C03663=1120.671,285.991,-75.029,-178.079,10.307,149.546
C03664=1120.667,286.239,-75.060,-178.076,10.310,149.546
C03665=1120.663,286.487,-75.091,-178.074,10.312,149.545
C03666=1120.659,286.735,-75.121,-178.070,10.314,149.545
C03667=1120.655,286.984,-75.152,-178.067,10.317,149.545
C03668=1120.650,287.231,-75.183,-178.064,10.319,149.545
C03669=1120.646,287.479,-75.215,-178.061,10.322,149.545
C03670=1120.643,287.727,-75.245,-178.058,10.325,149.545
C03671=1120.638,287.975,-75.276,-178.055,10.327,149.544
C03672=1120.634,288.224,-75.307,-178.052,10.330,149.544
C03673=1120.629,288.472,-75.338,-178.048,10.332,149.544
C03674=1120.625,288.719,-75.368,-178.045,10.335,149.544
C03675=1120.622,288.967,-75.400,-178.043,10.337,149.544
C03676=1120.617,289.215,-75.431,-178.040,10.340,149.544
C03677=1120.613,289.464,-75.462,-178.036,10.342,149.543
C03678=1120.608,289.712,-75.493,-178.034,10.345,149.543
C03679=1120.605,289.959,-75.523,-178.030,10.347,149.543
C03680=1120.601,290.208,-75.555,-178.027,10.350,149.543
C03681=1120.596,290.456,-75.585,-178.024,10.353,149.543
C03682=1120.593,290.704,-75.617,-178.021,10.355,149.542
C03683=1120.588,290.952,-75.648,-178.018,10.358,149.542
C03684=1120.584,291.200,-75.679,-178.015,10.360,149.542
C03685=1120.580,291.447,-75.710,-178.012,10.362,149.542
C03686=1120.576,291.696,-75.741,-178.009,10.365,149.542
C03687=1120.572,291.944,-75.772,-178.006,10.368,149.542
C03688=1120.568,292.192,-75.804,-178.003,10.370,149.541
C03689=1120.563,292.440,-75.834,-178.000,10.373,149.541
C03690=1120.559,292.689,-75.866,-177.997,10.375,149.541
C03691=1120.555,292.936,-75.897,-177.994,10.378,149.541
C03692=1120.551,293.185,-75.928,-177.991,10.381,149.541
C03693=1120.547,293.432,-75.960,-177.987,10.383,149.541
C03694=1120.544,293.645,-75.986,-177.985,10.385,149.540
C03695=1120.540,293.858,-76.013,-177.983,10.387,149.540
C03696=1120.536,294.071,-76.040,-177.979,10.390,149.540
C03697=1120.533,294.283,-76.067,-177.977,10.392,149.540
C03698=1120.529,294.497,-76.094,-177.975,10.394,149.540
C03699=1120.526,294.710,-76.121,-177.971,10.396,149.540
C03700=1120.522,294.923,-76.147,-177.969,10.398,149.539
C03701=1120.519,295.135,-76.174,-177.967,10.400,149.539
C03702=1120.515,295.383,-76.206,-177.964,10.402,149.539
C03703=1120.511,295.632,-76.237,-177.961,10.405,149.539
C03704=1120.507,295.879,-76.268,-177.957,10.408,149.539
C03705=1120.503,296.128,-76.300,-177.954,10.410,149.539
C03706=1120.498,296.375,-76.331,-177.951,10.413,149.539
C03707=1120.495,296.623,-76.363,-177.948,10.415,149.538
C03708=1120.490,296.871,-76.394,-177.945,10.418,149.538
C03709=1120.486,297.119,-76.426,-177.942,10.421,149.538
C03710=1120.482,297.367,-76.458,-177.939,10.423,149.538
C03711=1120.477,297.615,-76.489,-177.936,10.425,149.538
C03712=1120.474,297.863,-76.521,-177.933,10.428,149.537
C03713=1120.469,298.111,-76.552,-177.930,10.430,149.537
C03714=1120.466,298.359,-76.584,-177.927,10.433,149.537
C03715=1120.462,298.608,-76.615,-177.924,10.435,149.537
C03716=1120.457,298.855,-76.646,-177.921,10.438,149.537
C03717=1120.454,299.103,-76.678,-177.917,10.441,149.536
C03718=1120.448,299.351,-76.710,-177.914,10.443,149.536
C03719=1120.444,299.599,-76.742,-177.911,10.446,149.536
C03720=1120.441,299.847,-76.773,-177.908,10.449,149.536
C03721=1120.436,300.095,-76.805,-177.905,10.451,149.536
C03722=1120.433,300.343,-76.837,-177.903,10.453,149.536
C03723=1120.429,300.591,-76.869,-177.899,10.456,149.535
C03724=1120.424,300.838,-76.901,-177.896,10.458,149.535
C03725=1120.420,301.086,-76.932,-177.893,10.461,149.535
C03726=1120.416,301.335,-76.964,-177.890,10.463,149.535
C03727=1120.412,301.582,-76.995,-177.887,10.466,149.535
C03728=1120.408,301.831,-77.028,-177.884,10.469,149.535
C03729=1120.404,302.079,-77.059,-177.880,10.471,149.534
C03730=1120.400,302.326,-77.091,-177.877,10.474,149.534
C03731=1120.396,302.574,-77.123,-177.874,10.476,149.534
C03732=1120.391,302.822,-77.155,-177.871,10.479,149.534
C03733=1120.387,303.070,-77.187,-177.868,10.481,149.534
C03734=1120.383,303.318,-77.218,-177.865,10.483,149.533
C03735=1120.379,303.566,-77.251,-177.862,10.486,149.533
C03736=1120.375,303.814,-77.283,-177.859,10.488,149.533
C03737=1120.371,304.062,-77.314,-177.856,10.491,149.533
C03738=1120.366,304.310,-77.347,-177.853,10.494,149.533
C03739=1120.363,304.558,-77.379,-177.850,10.496,149.533
C03740=1120.359,304.805,-77.411,-177.846,10.499,149.532
C03741=1120.354,305.053,-77.443,-177.843,10.502,149.532
C03742=1120.351,305.301,-77.475,-177.840,10.504,149.532
C03743=1120.346,305.549,-77.507,-177.837,10.507,149.532
C03744=1120.342,305.797,-77.539,-177.834,10.509,149.532
C03745=1120.338,306.045,-77.571,-177.832,10.511,149.532
C03746=1120.334,306.293,-77.603,-177.828,10.514,149.531
C03747=1120.330,306.541,-77.636,-177.825,10.516,149.531
C03748=1120.326,306.789,-77.668,-177.822,10.519,149.531
C03749=1120.322,307.036,-77.700,-177.819,10.521,149.531
C03750=1120.318,307.249,-77.727,-177.816,10.523,149.531
C03751=1120.315,307.462,-77.754,-177.813,10.526,149.531
C03752=1120.311,307.675,-77.783,-177.811,10.528,149.530
C03753=1120.308,307.887,-77.811,-177.808,10.530,149.530
C03754=1120.304,308.100,-77.838,-177.805,10.532,149.530
C03755=1120.301,308.313,-77.865,-177.803,10.534,149.530
C03756=1120.297,308.526,-77.893,-177.800,10.537,149.530
C03757=1120.294,308.738,-77.921,-177.798,10.539,149.530
C03758=1120.290,308.986,-77.953,-177.794,10.541,149.529
C03759=1120.285,309.235,-77.986,-177.791,10.544,149.529
C03760=1120.282,309.482,-78.018,-177.788,10.546,149.529
C03761=1120.278,309.730,-78.051,-177.785,10.549,149.529
C03762=1120.274,309.978,-78.083,-177.782,10.552,149.529
C03763=1120.270,310.226,-78.116,-177.779,10.553,149.528
C03764=1120.265,310.474,-78.148,-177.776,10.556,149.528
C03765=1120.261,310.721,-78.180,-177.773,10.559,149.528
C03766=1120.257,310.970,-78.213,-177.770,10.561,149.528
C03767=1120.253,311.217,-78.245,-177.766,10.564,149.528
C03768=1120.249,311.465,-78.278,-177.764,10.567,149.528
C03769=1120.246,311.713,-78.310,-177.760,10.569,149.527
C03770=1120.241,311.961,-78.343,-177.757,10.571,149.527
C03771=1120.237,312.209,-78.376,-177.754,10.574,149.527
C03772=1120.233,312.457,-78.408,-177.751,10.577,149.527
C03773=1120.229,312.704,-78.441,-177.748,10.579,149.527
C03774=1120.224,312.952,-78.473,-177.744,10.582,149.526
C03775=1120.221,313.200,-78.506,-177.742,10.583,149.526
C03776=1120.217,313.447,-78.539,-177.739,10.586,149.526
C03777=1120.213,313.696,-78.571,-177.735,10.589,149.526
C03778=1120.209,313.943,-78.604,-177.733,10.591,149.526
C03779=1120.204,314.192,-78.636,-177.729,10.594,149.526
C03780=1120.201,314.439,-78.669,-177.726,10.597,149.525
C03781=1120.197,314.687,-78.702,-177.723,10.599,149.525
C03782=1120.192,314.935,-78.734,-177.720,10.602,149.525
C03783=1120.188,315.183,-78.767,-177.717,10.604,149.525
C03784=1120.185,315.430,-78.800,-177.713,10.607,149.525
C03785=1120.181,315.678,-78.833,-177.710,10.610,149.525
C03786=1120.176,315.926,-78.866,-177.707,10.612,149.524
C03787=1120.173,316.174,-78.898,-177.704,10.614,149.524
C03788=1120.169,316.421,-78.931,-177.701,10.616,149.524
C03789=1120.165,316.669,-78.965,-177.698,10.619,149.524
C03790=1120.160,316.918,-78.997,-177.695,10.621,149.523
C03791=1120.157,317.165,-79.030,-177.692,10.624,149.523
C03792=1120.153,317.413,-79.063,-177.689,10.627,149.523
C03793=1120.148,317.660,-79.096,-177.686,10.629,149.523
C03794=1120.144,317.908,-79.129,-177.682,10.632,149.523
C03795=1120.140,318.156,-79.162,-177.679,10.634,149.523
C03796=1120.136,318.404,-79.194,-177.676,10.637,149.522
C03797=1120.132,318.652,-79.227,-177.673,10.639,149.522
C03798=1120.128,318.899,-79.260,-177.670,10.642,149.522
C03799=1120.124,319.147,-79.293,-177.666,10.645,149.522
C03800=1120.120,319.395,-79.327,-177.664,10.646,149.522
C03801=1120.116,319.643,-79.360,-177.661,10.649,149.522
C03802=1120.112,319.891,-79.393,-177.658,10.652,149.521
C03803=1120.109,320.138,-79.426,-177.654,10.654,149.521
C03804=1120.105,320.386,-79.459,-177.651,10.657,149.521
C03805=1120.101,320.634,-79.492,-177.648,10.659,149.521
C03806=1120.097,320.847,-79.521,-177.646,10.661,149.521
C03807=1120.094,321.059,-79.549,-177.642,10.664,149.520
C03808=1120.090,321.272,-79.578,-177.640,10.666,149.520
C03809=1120.087,321.484,-79.607,-177.637,10.668,149.520
C03810=1120.083,321.698,-79.634,-177.634,10.670,149.520
C03811=1120.079,321.910,-79.663,-177.632,10.672,149.520
C03812=1120.077,322.122,-79.691,-177.629,10.674,149.520
C03813=1120.073,322.335,-79.720,-177.627,10.676,149.520
C03814=1120.069,322.583,-79.753,-177.623,10.679,149.519
C03815=1120.065,322.831,-79.786,-177.620,10.682,149.519
C03816=1120.061,323.078,-79.820,-177.617,10.684,149.519
C03817=1120.057,323.325,-79.853,-177.614,10.687,149.519
C03818=1120.053,323.574,-79.887,-177.611,10.689,149.519
C03819=1120.049,323.822,-79.920,-177.607,10.692,149.518
C03820=1120.045,324.069,-79.953,-177.604,10.694,149.518
C03821=1120.041,324.316,-79.987,-177.602,10.696,149.518
C03822=1120.037,324.564,-80.020,-177.598,10.699,149.518
C03823=1120.033,324.813,-80.054,-177.595,10.701,149.518
C03824=1120.029,325.060,-80.087,-177.592,10.704,149.518
C03825=1120.026,325.307,-80.121,-177.589,10.706,149.517
C03826=1120.021,325.555,-80.154,-177.586,10.709,149.517
C03827=1120.017,325.803,-80.187,-177.583,10.712,149.517
C03828=1120.014,326.051,-80.221,-177.579,10.714,149.517
C03829=1120.009,326.299,-80.255,-177.576,10.716,149.516
C03830=1120.005,326.547,-80.288,-177.573,10.719,149.516
C03831=1120.001,326.794,-80.321,-177.570,10.722,149.516
C03832=1119.997,327.041,-80.355,-177.566,10.724,149.516
C03833=1119.993,327.290,-80.389,-177.563,10.727,149.516
C03834=1119.990,327.537,-80.423,-177.561,10.729,149.516
C03835=1119.986,327.785,-80.456,-177.557,10.731,149.515
C03836=1119.981,328.033,-80.490,-177.555,10.734,149.515
C03837=1119.977,328.280,-80.524,-177.551,10.736,149.515
C03838=1119.973,328.528,-80.557,-177.548,10.739,149.515
C03839=1119.969,328.775,-80.591,-177.545,10.741,149.515
C03840=1119.965,329.023,-80.624,-177.542,10.744,149.514
C03841=1119.961,329.271,-80.659,-177.538,10.746,149.514
C03842=1119.957,329.519,-80.692,-177.535,10.749,149.514
C03843=1119.953,329.766,-80.726,-177.532,10.752,149.514
C03844=1119.950,330.014,-80.759,-177.529,10.754,149.514
C03845=1119.945,330.262,-80.794,-177.525,10.757,149.513
C03846=1119.941,330.509,-80.828,-177.523,10.759,149.513
C03847=1119.937,330.757,-80.861,-177.519,10.762,149.513
C03848=1119.934,331.005,-80.895,-177.517,10.763,149.513
C03849=1119.929,331.253,-80.929,-177.513,10.766,149.513
C03850=1119.925,331.500,-80.963,-177.510,10.769,149.513
C03851=1119.922,331.747,-80.997,-177.507,10.771,149.512
C03852=1119.918,331.995,-81.030,-177.504,10.774,149.512
C03853=1119.913,332.243,-81.065,-177.501,10.776,149.512
C03854=1119.910,332.490,-81.099,-177.497,10.779,149.512
C03855=1119.906,332.738,-81.132,-177.494,10.781,149.512
C03856=1119.902,332.986,-81.167,-177.491,10.784,149.511
C03857=1119.898,333.233,-81.201,-177.488,10.786,149.511
C03858=1119.893,333.481,-81.234,-177.485,10.789,149.511
C03859=1119.890,333.729,-81.269,-177.481,10.791,149.511
C03860=1119.886,333.976,-81.303,-177.478,10.794,149.511
C03861=1119.882,334.224,-81.337,-177.475,10.797,149.510
C03862=1119.878,334.437,-81.366,-177.472,10.798,149.510
C03863=1119.875,334.649,-81.395,-177.470,10.800,149.510
C03864=1119.872,334.861,-81.425,-177.467,10.803,149.510
C03865=1119.868,335.074,-81.454,-177.464,10.805,149.510
C03866=1119.865,335.286,-81.484,-177.462,10.806,149.510
C03867=1119.862,335.499,-81.512,-177.459,10.809,149.509
C03868=1119.858,335.711,-81.542,-177.456,10.811,149.509
C03869=1119.855,335.924,-81.572,-177.454,10.813,149.509
C03870=1119.852,336.172,-81.605,-177.450,10.815,149.509
C03871=1119.847,336.420,-81.640,-177.447,10.818,149.509
C03872=1119.843,336.667,-81.673,-177.444,10.820,149.508
C03873=1119.839,336.915,-81.708,-177.441,10.823,149.508
C03874=1119.835,337.162,-81.742,-177.438,10.825,149.508
C03875=1119.831,337.410,-81.777,-177.434,10.828,149.508
C03876=1119.828,337.657,-81.811,-177.431,10.830,149.508
C03877=1119.824,337.905,-81.846,-177.428,10.833,149.508
C03878=1119.820,338.152,-81.880,-177.425,10.836,149.507
C03879=1119.816,338.400,-81.914,-177.421,10.838,149.507
C03880=1119.812,338.648,-81.948,-177.418,10.841,149.507
C03881=1119.808,338.896,-81.983,-177.415,10.843,149.507
C03882=1119.804,339.143,-82.017,-177.412,10.846,149.507
C03883=1119.800,339.391,-82.052,-177.409,10.847,149.506
C03884=1119.796,339.638,-82.086,-177.406,10.850,149.506
C03885=1119.793,339.886,-82.121,-177.403,10.852,149.506
C03886=1119.788,340.133,-82.156,-177.400,10.855,149.506
C03887=1119.784,340.381,-82.191,-177.396,10.858,149.506
C03888=1119.780,340.628,-82.224,-177.393,10.860,149.505
C03889=1119.776,340.876,-82.259,-177.390,10.863,149.505
C03890=1119.773,341.123,-82.293,-177.386,10.865,149.505
C03891=1119.769,341.371,-82.329,-177.383,10.868,149.505
C03892=1119.764,341.618,-82.363,-177.380,10.870,149.505
C03893=1119.761,341.866,-82.397,-177.377,10.873,149.504
C03894=1119.756,342.114,-82.432,-177.374,10.875,149.504
C03895=1119.753,342.362,-82.467,-177.370,10.878,149.504
C03896=1119.748,342.608,-82.502,-177.367,10.880,149.504
C03897=1119.745,342.856,-82.536,-177.364,10.883,149.504
C03898=1119.740,343.104,-82.571,-177.361,10.885,149.503
C03899=1119.737,343.351,-82.606,-177.358,10.887,149.503
C03900=1119.734,343.599,-82.640,-177.355,10.889,149.503
C03901=1119.729,343.846,-82.675,-177.352,10.892,149.503
C03902=1119.725,344.094,-82.710,-177.348,10.895,149.503
C03903=1119.721,344.341,-82.745,-177.345,10.897,149.502
C03904=1119.718,344.589,-82.779,-177.342,10.900,149.502
C03905=1119.714,344.837,-82.815,-177.338,10.902,149.502
C03906=1119.709,345.084,-82.849,-177.335,10.904,149.502
C03907=1119.706,345.332,-82.885,-177.332,10.907,149.502
C03908=1119.701,345.579,-82.919,-177.329,10.910,149.501
C03909=1119.698,345.826,-82.954,-177.326,10.912,149.501
C03910=1119.694,346.074,-82.989,-177.322,10.915,149.501
C03911=1119.690,346.322,-83.023,-177.319,10.917,149.501
C03912=1119.686,346.569,-83.059,-177.316,10.919,149.500
C03913=1119.682,346.817,-83.094,-177.313,10.922,149.500
C03914=1119.678,347.064,-83.129,-177.310,10.924,149.500
C03915=1119.675,347.311,-83.164,-177.307,10.927,149.500
C03916=1119.671,347.559,-83.199,-177.303,10.929,149.500
C03917=1119.667,347.806,-83.234,-177.300,10.931,149.500
C03918=1119.663,348.020,-83.264,-177.298,10.933,149.499
C03919=1119.660,348.232,-83.294,-177.295,10.936,149.499
C03920=1119.657,348.444,-83.324,-177.292,10.938,149.499
C03921=1119.653,348.656,-83.355,-177.289,10.940,149.499
C03922=1119.650,348.868,-83.384,-177.286,10.942,149.499
C03923=1119.646,349.081,-83.414,-177.284,10.944,149.499
C03924=1119.644,349.293,-83.445,-177.281,10.947,149.498
C03925=1119.640,349.506,-83.475,-177.278,10.948,149.498
C03926=1119.636,349.753,-83.511,-177.275,10.951,149.498
C03927=1119.631,350.001,-83.545,-177.271,10.954,149.498
C03928=1119.628,350.248,-83.581,-177.267,10.956,149.497
C03929=1119.624,350.496,-83.616,-177.264,10.959,149.497
C03930=1119.621,350.743,-83.651,-177.261,10.961,149.497
C03931=1119.617,350.990,-83.686,-177.258,10.964,149.497
C03932=1119.613,351.238,-83.721,-177.254,10.966,149.497
C03933=1119.609,351.485,-83.757,-177.250,10.969,149.496
C03934=1119.606,351.733,-83.792,-177.247,10.972,149.496
C03935=1119.601,351.980,-83.828,-177.243,10.974,149.496
C03936=1119.597,352.228,-83.863,-177.240,10.977,149.495
C03937=1119.593,352.475,-83.899,-177.237,10.979,149.495
C03938=1119.589,352.723,-83.934,-177.233,10.981,149.495
C03939=1119.586,352.970,-83.970,-177.229,10.985,149.495
C03940=1119.581,353.217,-84.005,-177.226,10.987,149.495
C03941=1119.578,353.465,-84.040,-177.222,10.989,149.494
C03942=1119.574,353.712,-84.076,-177.219,10.992,149.494
C03943=1119.570,353.960,-84.111,-177.216,10.994,149.494
C03944=1119.567,354.207,-84.147,-177.212,10.997,149.494
C03945=1119.563,354.454,-84.182,-177.209,10.999,149.493
C03946=1119.559,354.702,-84.218,-177.206,11.002,149.493
C03947=1119.555,354.949,-84.253,-177.202,11.004,149.493
C03948=1119.551,355.197,-84.289,-177.198,11.007,149.493
C03949=1119.547,355.444,-84.325,-177.195,11.009,149.492
C03950=1119.543,355.692,-84.361,-177.192,11.012,149.492
C03951=1119.540,355.939,-84.396,-177.188,11.014,149.492
C03952=1119.536,356.186,-84.431,-177.185,11.017,149.491
C03953=1119.532,356.434,-84.467,-177.181,11.019,149.491
C03954=1119.527,356.681,-84.503,-177.178,11.021,149.491
C03955=1119.524,356.929,-84.538,-177.175,11.024,149.491
C03956=1119.520,357.176,-84.574,-177.171,11.026,149.491
C03957=1119.517,357.423,-84.610,-177.168,11.029,149.490
C03958=1119.513,357.671,-84.646,-177.164,11.031,149.490
C03959=1119.509,357.919,-84.682,-177.161,11.033,149.490
C03960=1119.505,358.166,-84.718,-177.158,11.036,149.490
C03961=1119.501,358.414,-84.753,-177.154,11.038,149.489
C03962=1119.498,358.661,-84.789,-177.151,11.041,149.489
C03963=1119.494,358.908,-84.825,-177.147,11.043,149.489
C03964=1119.489,359.155,-84.861,-177.144,11.045,149.488
C03965=1119.486,359.403,-84.896,-177.141,11.048,149.488
C03966=1119.482,359.650,-84.932,-177.137,11.050,149.488
C03967=1119.478,359.897,-84.969,-177.134,11.053,149.488
C03968=1119.474,360.145,-85.004,-177.130,11.055,149.487
C03969=1119.471,360.392,-85.040,-177.127,11.057,149.487
C03970=1119.467,360.640,-85.077,-177.123,11.060,149.487
C03971=1119.463,360.887,-85.112,-177.120,11.062,149.487
C03972=1119.460,361.134,-85.148,-177.117,11.065,149.486
C03973=1119.455,361.382,-85.185,-177.114,11.067,149.486
C03974=1119.452,361.594,-85.216,-177.110,11.069,149.486
C03975=1119.449,361.806,-85.246,-177.108,11.071,149.486
C03976=1119.446,362.019,-85.277,-177.104,11.074,149.485
C03977=1119.442,362.231,-85.308,-177.102,11.075,149.485
C03978=1119.439,362.443,-85.339,-177.098,11.078,149.485
C03979=1119.436,362.655,-85.370,-177.096,11.079,149.485
C03980=1119.433,362.867,-85.401,-177.093,11.081,149.485
C03981=1119.430,363.079,-85.432,-177.090,11.084,149.484
C03982=1119.426,363.327,-85.469,-177.086,11.086,149.484
C03983=1119.422,363.574,-85.505,-177.083,11.089,149.484
C03984=1119.418,363.821,-85.541,-177.080,11.091,149.484
C03985=1119.415,364.068,-85.578,-177.076,11.094,149.483
C03986=1119.411,364.316,-85.613,-177.073,11.096,149.483
C03987=1119.407,364.563,-85.650,-177.070,11.097,149.483
C03988=1119.403,364.810,-85.686,-177.067,11.100,149.483
C03989=1119.399,365.058,-85.722,-177.063,11.102,149.482
C03990=1119.396,365.304,-85.759,-177.060,11.105,149.482
C03991=1119.392,365.553,-85.795,-177.057,11.107,149.482
C03992=1119.389,365.800,-85.831,-177.054,11.110,149.482
C03993=1119.385,366.047,-85.868,-177.050,11.112,149.481
C03994=1119.380,366.295,-85.904,-177.047,11.114,149.481
C03995=1119.377,366.542,-85.941,-177.043,11.117,149.481
C03996=1119.373,366.789,-85.978,-177.040,11.119,149.481
C03997=1119.369,367.036,-86.014,-177.037,11.122,149.480
C03998=1119.365,367.284,-86.050,-177.033,11.124,149.480
C03999=1119.362,367.531,-86.086,-177.030,11.126,149.480
C04000=1119.357,367.778,-86.123,-177.026,11.129,149.480
C04001=1119.354,368.026,-86.160,-177.024,11.131,149.479
C04002=1119.350,368.273,-86.196,-177.020,11.133,149.479
C04003=1119.346,368.520,-86.233,-177.017,11.136,149.479
C04004=1119.342,368.768,-86.270,-177.014,11.138,149.479
C04005=1119.339,369.014,-86.306,-177.010,11.140,149.479
C04006=1119.335,369.262,-86.343,-177.007,11.143,149.478
C04007=1119.332,369.509,-86.379,-177.004,11.145,149.478
C04008=1119.328,369.756,-86.416,-177.001,11.148,149.478
C04009=1119.324,370.004,-86.453,-176.997,11.150,149.478
C04010=1119.320,370.250,-86.489,-176.994,11.153,149.477
C04011=1119.316,370.498,-86.525,-176.990,11.155,149.477
C04012=1119.312,370.745,-86.562,-176.988,11.157,149.477
C04013=1119.308,370.993,-86.600,-176.984,11.159,149.477
C04014=1119.305,371.240,-86.636,-176.981,11.162,149.476
C04015=1119.301,371.487,-86.673,-176.978,11.164,149.476
C04016=1119.297,371.735,-86.710,-176.974,11.167,149.476
C04017=1119.294,371.982,-86.746,-176.971,11.169,149.476
C04018=1119.290,372.229,-86.783,-176.968,11.172,149.476
C04019=1119.286,372.476,-86.821,-176.964,11.174,149.475
C04020=1119.282,372.723,-86.857,-176.961,11.177,149.475
C04021=1119.279,372.971,-86.894,-176.959,11.178,149.475
C04022=1119.275,373.218,-86.931,-176.955,11.181,149.475
C04023=1119.271,373.465,-86.968,-176.952,11.183,149.475
C04024=1119.267,373.712,-87.005,-176.949,11.186,149.475
C04025=1119.264,373.960,-87.042,-176.946,11.188,149.474
C04026=1119.260,374.207,-87.078,-176.942,11.191,149.474
C04027=1119.256,374.454,-87.116,-176.939,11.193,149.474
C04028=1119.252,374.701,-87.153,-176.936,11.196,149.474
C04029=1119.249,374.949,-87.190,-176.933,11.198,149.473
C04030=1119.245,375.160,-87.221,-176.930,11.200,149.473
C04031=1119.242,375.373,-87.253,-176.928,11.202,149.473
C04032=1119.239,375.585,-87.285,-176.925,11.204,149.473
C04033=1119.236,375.796,-87.317,-176.922,11.207,149.473
C04034=1119.233,376.009,-87.348,-176.919,11.208,149.473
C04035=1119.230,376.221,-87.380,-176.917,11.210,149.473
C04036=1119.226,376.433,-87.412,-176.914,11.213,149.472
C04037=1119.223,376.645,-87.444,-176.911,11.215,149.472
C04038=1119.219,376.892,-87.481,-176.908,11.217,149.472
C04039=1119.215,377.140,-87.518,-176.905,11.220,149.472
C04040=1119.212,377.386,-87.556,-176.902,11.222,149.472
C04041=1119.208,377.633,-87.593,-176.898,11.225,149.472
C04042=1119.204,377.881,-87.630,-176.896,11.227,149.472
C04043=1119.200,378.128,-87.668,-176.893,11.229,149.471
C04044=1119.196,378.375,-87.705,-176.889,11.232,149.471
C04045=1119.194,378.622,-87.742,-176.886,11.234,149.471
C04046=1119.190,378.869,-87.779,-176.883,11.237,149.471
C04047=1119.186,379.116,-87.816,-176.880,11.240,149.471
C04048=1119.182,379.364,-87.854,-176.877,11.242,149.471
C04049=1119.178,379.611,-87.890,-176.874,11.245,149.471
C04050=1119.175,379.858,-87.928,-176.871,11.247,149.470
C04051=1119.170,380.106,-87.966,-176.868,11.249,149.470
C04052=1119.166,380.352,-88.003,-176.865,11.252,149.470
C04053=1119.163,380.600,-88.041,-176.862,11.254,149.470
C04054=1119.159,380.847,-88.078,-176.859,11.257,149.470
C04055=1119.156,381.094,-88.116,-176.855,11.260,149.470
C04056=1119.152,381.341,-88.153,-176.853,11.262,149.470
C04057=1119.148,381.588,-88.191,-176.849,11.265,149.469
C04058=1119.145,381.836,-88.228,-176.847,11.267,149.469
C04059=1119.141,382.082,-88.265,-176.844,11.269,149.469
C04060=1119.138,382.330,-88.303,-176.841,11.272,149.469
C04061=1119.134,382.577,-88.340,-176.837,11.275,149.469
C04062=1119.130,382.824,-88.378,-176.835,11.278,149.469
C04063=1119.127,383.071,-88.416,-176.832,11.280,149.469
C04064=1119.122,383.319,-88.453,-176.828,11.283,149.469
C04065=1119.119,383.565,-88.491,-176.826,11.285,149.469
C04066=1119.115,383.812,-88.529,-176.824,11.287,149.469
C04067=1119.111,384.060,-88.566,-176.822,11.289,149.469
C04068=1119.107,384.306,-88.603,-176.820,11.291,149.469
C04069=1119.104,384.554,-88.641,-176.818,11.294,149.469
C04070=1119.101,384.800,-88.679,-176.816,11.296,149.469
C04071=1119.096,385.048,-88.717,-176.813,11.299,149.469
C04072=1119.092,385.295,-88.754,-176.811,11.301,149.469
C04073=1119.089,385.542,-88.792,-176.809,11.303,149.469
C04074=1119.086,385.789,-88.830,-176.807,11.305,149.469
C04075=1119.082,386.036,-88.868,-176.805,11.308,149.469
C04076=1119.077,386.284,-88.905,-176.803,11.310,149.469
C04077=1119.074,386.531,-88.943,-176.801,11.312,149.469
C04078=1119.071,386.777,-88.981,-176.799,11.314,149.469
C04079=1119.067,387.025,-89.019,-176.797,11.317,149.470
C04080=1119.064,387.272,-89.057,-176.794,11.320,149.470
C04081=1119.060,387.519,-89.095,-176.792,11.322,149.470
C04082=1119.056,387.767,-89.132,-176.790,11.324,149.470
C04083=1119.052,388.013,-89.170,-176.788,11.327,149.470
C04084=1119.049,388.261,-89.208,-176.786,11.329,149.470
C04085=1119.045,388.507,-89.246,-176.784,11.332,149.470
C04086=1119.042,388.719,-89.278,-176.783,11.334,149.470
C04087=1119.039,388.931,-89.311,-176.781,11.336,149.470
C04088=1119.036,389.143,-89.343,-176.779,11.338,149.471
C04089=1119.032,389.356,-89.376,-176.777,11.341,149.471
C04090=1119.030,389.567,-89.408,-176.776,11.343,149.471
C04091=1119.026,389.779,-89.441,-176.774,11.345,149.471
C04092=1119.023,389.990,-89.474,-176.773,11.347,149.471
C04093=1119.020,390.202,-89.506,-176.771,11.350,149.471
C04094=1119.017,390.450,-89.544,-176.769,11.352,149.472
C04095=1119.012,390.696,-89.582,-176.767,11.356,149.472
C04096=1119.009,390.944,-89.620,-176.765,11.358,149.472
C04097=1119.005,391.190,-89.657,-176.763,11.361,149.472
C04098=1119.001,391.438,-89.696,-176.761,11.364,149.473
C04099=1118.998,391.685,-89.734,-176.759,11.367,149.473
C04100=1118.994,391.932,-89.771,-176.758,11.369,149.473
C04101=1118.991,392.179,-89.810,-176.755,11.372,149.473
C04102=1118.987,392.427,-89.848,-176.754,11.375,149.474
C04103=1118.984,392.673,-89.886,-176.752,11.378,149.474
C04104=1118.980,392.920,-89.925,-176.750,11.381,149.474
C04105=1118.976,393.167,-89.962,-176.748,11.384,149.475
C04106=1118.972,393.414,-90.001,-176.746,11.387,149.475
C04107=1118.969,393.662,-90.039,-176.745,11.390,149.475
C04108=1118.965,393.908,-90.076,-176.743,11.393,149.476
C04109=1118.961,394.156,-90.115,-176.741,11.396,149.476
C04110=1118.958,394.403,-90.153,-176.740,11.399,149.476
C04111=1118.954,394.649,-90.192,-176.738,11.402,149.477
C04112=1118.951,394.896,-90.230,-176.737,11.405,149.477
C04113=1118.946,395.143,-90.268,-176.734,11.409,149.478
C04114=1118.943,395.391,-90.306,-176.732,11.412,149.478
C04115=1118.940,395.637,-90.344,-176.731,11.415,149.478
C04116=1118.936,395.884,-90.383,-176.729,11.418,149.479
C04117=1118.932,396.131,-90.421,-176.728,11.421,149.479
C04118=1118.929,396.379,-90.459,-176.726,11.425,149.480
C04119=1118.925,396.625,-90.497,-176.724,11.428,149.480
C04120=1118.921,396.873,-90.536,-176.723,11.431,149.481
C04121=1118.918,397.120,-90.574,-176.721,11.435,149.481
C04122=1118.914,397.367,-90.612,-176.720,11.438,149.481
C04123=1118.911,397.613,-90.651,-176.718,11.442,149.482
C04124=1118.907,397.861,-90.689,-176.716,11.445,149.482
C04125=1118.903,398.108,-90.727,-176.715,11.448,149.483
C04126=1118.899,398.354,-90.766,-176.713,11.452,149.483
C04127=1118.896,398.602,-90.804,-176.711,11.456,149.484
C04128=1118.892,398.849,-90.843,-176.710,11.459,149.484
C04129=1118.889,399.096,-90.881,-176.708,11.463,149.485
C04130=1118.885,399.343,-90.919,-176.707,11.466,149.486
C04131=1118.881,399.590,-90.959,-176.706,11.469,149.486
C04132=1118.878,399.837,-90.997,-176.704,11.473,149.487
C04133=1118.874,400.083,-91.035,-176.703,11.477,149.487
C04134=1118.870,400.331,-91.073,-176.701,11.481,149.488
C04135=1118.867,400.578,-91.113,-176.699,11.485,149.488
C04136=1118.864,400.825,-91.151,-176.698,11.488,149.489
C04137=1118.859,401.072,-91.189,-176.697,11.492,149.490
C04138=1118.856,401.319,-91.228,-176.695,11.496,149.490
C04139=1118.852,401.566,-91.266,-176.694,11.500,149.491
C04140=1118.849,401.813,-91.305,-176.692,11.504,149.492
C04141=1118.846,402.060,-91.344,-176.691,11.508,149.492
C04142=1118.842,402.272,-91.376,-176.690,11.511,149.493
C04143=1118.839,402.484,-91.410,-176.689,11.514,149.493
C04144=1118.836,402.695,-91.443,-176.687,11.518,149.494
C04145=1118.833,402.907,-91.476,-176.686,11.521,149.495
C04146=1118.830,403.119,-91.510,-176.685,11.525,149.495
C04147=1118.827,403.330,-91.542,-176.684,11.528,149.496
C04148=1118.824,403.542,-91.576,-176.683,11.532,149.497
C04149=1118.821,403.754,-91.609,-176.681,11.536,149.497
C04150=1118.816,404.000,-91.647,-176.681,11.540,149.498
C04151=1118.813,404.247,-91.686,-176.679,11.544,149.499
C04152=1118.810,404.494,-91.725,-176.678,11.548,149.500
C04153=1118.806,404.742,-91.764,-176.677,11.552,149.500
C04154=1118.802,404.989,-91.803,-176.676,11.557,149.501
C04155=1118.799,405.235,-91.841,-176.674,11.561,149.502
C04156=1118.795,405.482,-91.880,-176.673,11.565,149.503
C04157=1118.791,405.729,-91.919,-176.672,11.570,149.504
C04158=1118.788,405.976,-91.958,-176.671,11.574,149.505
C04159=1118.784,406.223,-91.996,-176.669,11.579,149.505
C04160=1118.781,406.470,-92.035,-176.668,11.583,149.506
C04161=1118.777,406.717,-92.075,-176.667,11.588,149.507
C04162=1118.774,406.963,-92.113,-176.666,11.592,149.508
C04163=1118.770,407.211,-92.151,-176.665,11.597,149.509
C04164=1118.766,407.458,-92.191,-176.664,11.602,149.510
C04165=1118.763,407.705,-92.230,-176.663,11.606,149.511
C04166=1118.760,407.951,-92.269,-176.662,11.611,149.512
C04167=1118.756,408.198,-92.308,-176.661,11.615,149.513
C04168=1118.752,408.446,-92.346,-176.659,11.620,149.514
C04169=1118.749,408.693,-92.386,-176.659,11.625,149.515
C04170=1118.746,408.940,-92.424,-176.658,11.630,149.516
C04171=1118.741,409.186,-92.463,-176.657,11.635,149.517
C04172=1118.738,409.433,-92.502,-176.656,11.640,149.518
C04173=1118.734,409.680,-92.542,-176.655,11.644,149.519
C04174=1118.731,409.927,-92.581,-176.654,11.650,149.520
C04175=1118.727,410.174,-92.620,-176.653,11.654,149.521
C04176=1118.724,410.420,-92.659,-176.652,11.659,149.522
C04177=1118.720,410.668,-92.697,-176.651,11.665,149.523
C04178=1118.717,410.915,-92.737,-176.650,11.669,149.524
C04179=1118.713,411.162,-92.776,-176.649,11.675,149.525
C04180=1118.709,411.409,-92.815,-176.648,11.680,149.527
C04181=1118.706,411.656,-92.854,-176.648,11.685,149.528
C04182=1118.702,411.903,-92.894,-176.647,11.690,149.529
C04183=1118.699,412.149,-92.932,-176.646,11.696,149.530
C04184=1118.696,412.396,-92.971,-176.645,11.701,149.531
C04185=1118.692,412.643,-93.011,-176.645,11.706,149.533
C04186=1118.688,412.890,-93.050,-176.643,11.712,149.534
C04187=1118.684,413.136,-93.089,-176.643,11.717,149.535
C04188=1118.681,413.383,-93.129,-176.642,11.723,149.536
C04189=1118.677,413.630,-93.168,-176.642,11.728,149.537
C04190=1118.675,413.877,-93.207,-176.641,11.734,149.539
C04191=1118.671,414.124,-93.246,-176.640,11.739,149.540
C04192=1118.670,414.371,-93.285,-176.640,11.744,149.541
C04193=1118.668,414.618,-93.324,-176.639,11.750,149.543
C04194=1118.667,414.864,-93.364,-176.638,11.756,149.544
C04195=1118.666,415.112,-93.402,-176.637,11.762,149.545
C04196=1118.666,415.359,-93.441,-176.637,11.767,149.547
C04197=1118.667,415.606,-93.480,-176.636,11.773,149.548
C04198=1118.668,415.818,-93.513,-176.636,11.778,149.549
C04199=1118.669,416.028,-93.546,-176.636,11.783,149.550
C04200=1118.671,416.240,-93.579,-176.635,11.788,149.552
C04201=1118.673,416.452,-93.612,-176.635,11.793,149.553
C04202=1118.675,416.663,-93.645,-176.635,11.798,149.554
C04203=1118.678,416.875,-93.678,-176.634,11.803,149.555
C04204=1118.682,417.086,-93.711,-176.634,11.808,149.556
C04205=1118.686,417.298,-93.744,-176.634,11.813,149.558
C04206=1118.267,417.298,-93.806,-176.626,11.818,149.557
C04207=1118.263,417.086,-93.774,-176.626,11.813,149.556
C04208=1118.259,416.874,-93.741,-176.627,11.807,149.555
C04209=1118.256,416.663,-93.708,-176.627,11.802,149.553
C04210=1118.254,416.452,-93.675,-176.628,11.797,149.552
C04211=1118.252,416.240,-93.642,-176.628,11.792,149.551
C04212=1118.250,416.028,-93.609,-176.628,11.787,149.550
C04213=1118.249,415.818,-93.576,-176.629,11.782,149.549
C04214=1118.248,415.605,-93.542,-176.629,11.777,149.547
C04215=1118.248,415.359,-93.503,-176.630,11.772,149.546
C04216=1118.247,415.112,-93.465,-176.631,11.766,149.545
C04217=1118.247,414.865,-93.426,-176.632,11.760,149.543
C04218=1118.249,414.618,-93.387,-176.632,11.755,149.542
C04219=1118.250,414.370,-93.347,-176.633,11.749,149.541
C04220=1118.252,414.124,-93.309,-176.633,11.743,149.539
C04221=1118.255,413.877,-93.269,-176.634,11.737,149.538
C04222=1118.258,413.630,-93.230,-176.635,11.732,149.537
C04223=1118.262,413.383,-93.191,-176.636,11.726,149.536
C04224=1118.265,413.136,-93.152,-176.636,11.721,149.534
C04225=1118.269,412.890,-93.112,-176.637,11.716,149.533
C04226=1118.272,412.643,-93.073,-176.638,11.710,149.532
C04227=1118.276,412.396,-93.034,-176.639,11.704,149.531
C04228=1118.280,412.149,-92.995,-176.640,11.700,149.530
C04229=1118.283,411.902,-92.955,-176.641,11.694,149.528
C04230=1118.287,411.655,-92.916,-176.641,11.689,149.527
C04231=1118.290,411.408,-92.877,-176.643,11.684,149.526
C04232=1118.293,411.161,-92.838,-176.644,11.678,149.525
C04233=1118.297,410.914,-92.799,-176.644,11.673,149.524
C04234=1118.301,410.667,-92.760,-176.645,11.668,149.523
C04235=1118.304,410.420,-92.720,-176.646,11.663,149.522
C04236=1118.308,410.173,-92.681,-176.647,11.658,149.520
C04237=1118.312,409.927,-92.642,-176.648,11.653,149.520
C04238=1118.315,409.680,-92.604,-176.649,11.648,149.518
C04239=1118.319,409.433,-92.564,-176.650,11.643,149.517
C04240=1118.322,409.186,-92.525,-176.651,11.638,149.516
C04241=1118.326,408.939,-92.486,-176.652,11.633,149.515
C04242=1118.329,408.692,-92.447,-176.653,11.628,149.514
C04243=1118.333,408.445,-92.409,-176.655,11.623,149.513
C04244=1118.336,408.198,-92.369,-176.656,11.619,149.512
C04245=1118.340,407.951,-92.330,-176.657,11.614,149.511
C04246=1118.343,407.704,-92.291,-176.658,11.609,149.510
C04247=1118.347,407.457,-92.252,-176.659,11.605,149.510
C04248=1118.351,407.211,-92.213,-176.660,11.600,149.509
C04249=1118.355,406.964,-92.175,-176.661,11.596,149.508
C04250=1118.358,406.717,-92.136,-176.663,11.590,149.507
C04251=1118.362,406.470,-92.096,-176.663,11.586,149.506
C04252=1118.365,406.223,-92.058,-176.665,11.582,149.505
C04253=1118.369,405.976,-92.019,-176.666,11.577,149.504
C04254=1118.372,405.729,-91.980,-176.667,11.573,149.503
C04255=1118.376,405.482,-91.941,-176.669,11.568,149.502
C04256=1118.379,405.236,-91.902,-176.670,11.564,149.502
C04257=1118.383,404.988,-91.864,-176.671,11.560,149.501
C04258=1118.387,404.741,-91.825,-176.672,11.555,149.500
C04259=1118.390,404.495,-91.786,-176.673,11.551,149.499
C04260=1118.394,404.247,-91.747,-176.675,11.547,149.498
C04261=1118.398,404.001,-91.709,-176.676,11.543,149.498
C04262=1118.401,403.754,-91.670,-176.677,11.539,149.497
C04263=1118.404,403.542,-91.637,-176.679,11.534,149.496
C04264=1118.407,403.331,-91.603,-176.680,11.531,149.496
C04265=1118.411,403.118,-91.571,-176.681,11.527,149.495
C04266=1118.414,402.907,-91.537,-176.682,11.524,149.494
C04267=1118.417,402.695,-91.504,-176.683,11.520,149.494
C04268=1118.419,402.484,-91.471,-176.684,11.517,149.493
C04269=1118.422,402.272,-91.438,-176.686,11.514,149.493
C04270=1118.426,402.060,-91.405,-176.687,11.510,149.492
C04271=1118.429,401.813,-91.366,-176.689,11.506,149.491
C04272=1118.432,401.566,-91.328,-176.690,11.502,149.491
C04273=1118.436,401.319,-91.288,-176.691,11.498,149.490
C04274=1118.441,401.072,-91.250,-176.693,11.494,149.489
C04275=1118.443,400.825,-91.211,-176.694,11.491,149.489
C04276=1118.447,400.578,-91.173,-176.695,11.487,149.488
C04277=1118.450,400.331,-91.134,-176.697,11.483,149.488
C04278=1118.455,400.084,-91.096,-176.699,11.479,149.487
C04279=1118.459,399.837,-91.058,-176.700,11.475,149.486
C04280=1118.462,399.590,-91.019,-176.702,11.472,149.486
C04281=1118.466,399.342,-90.980,-176.703,11.469,149.485
C04282=1118.469,399.097,-90.942,-176.705,11.465,149.485
C04283=1118.473,398.849,-90.904,-176.706,11.461,149.484
C04284=1118.476,398.602,-90.865,-176.708,11.457,149.484
C04285=1118.480,398.355,-90.826,-176.709,11.454,149.483
C04286=1118.484,398.108,-90.789,-176.711,11.451,149.483
C04287=1118.487,397.861,-90.750,-176.713,11.447,149.482
C04288=1118.490,397.614,-90.712,-176.715,11.443,149.482
C04289=1118.495,397.367,-90.673,-176.716,11.440,149.481
C04290=1118.498,397.120,-90.635,-176.718,11.437,149.481
C04291=1118.502,396.873,-90.596,-176.720,11.433,149.480
C04292=1118.505,396.626,-90.559,-176.721,11.430,149.480
C04293=1118.509,396.379,-90.519,-176.723,11.426,149.479
C04294=1118.512,396.132,-90.482,-176.725,11.423,149.479
C04295=1118.517,395.885,-90.443,-176.726,11.420,149.478
C04296=1118.520,395.638,-90.405,-176.728,11.416,149.478
C04297=1118.524,395.391,-90.366,-176.730,11.414,149.478
C04298=1118.527,395.144,-90.329,-176.732,11.410,149.477
C04299=1118.531,394.897,-90.290,-176.733,11.406,149.477
C04300=1118.535,394.649,-90.252,-176.735,11.404,149.476
C04301=1118.539,394.403,-90.213,-176.737,11.400,149.476
C04302=1118.542,394.156,-90.175,-176.739,11.398,149.476
C04303=1118.545,393.909,-90.137,-176.741,11.394,149.475
C04304=1118.550,393.662,-90.099,-176.742,11.391,149.475
C04305=1118.553,393.414,-90.061,-176.744,11.388,149.475
C04306=1118.557,393.167,-90.023,-176.746,11.385,149.474
C04307=1118.561,392.920,-89.985,-176.748,11.382,149.474
C04308=1118.563,392.674,-89.946,-176.750,11.379,149.474
C04309=1118.568,392.427,-89.908,-176.751,11.377,149.473
C04310=1118.571,392.180,-89.870,-176.753,11.373,149.473
C04311=1118.574,391.932,-89.832,-176.755,11.371,149.473
C04312=1118.579,391.685,-89.794,-176.757,11.367,149.473
C04313=1118.582,391.438,-89.756,-176.759,11.365,149.472
C04314=1118.585,391.191,-89.718,-176.761,11.362,149.472
C04315=1118.590,390.944,-89.680,-176.763,11.359,149.472
C04316=1118.593,390.697,-89.642,-176.765,11.357,149.472
C04317=1118.597,390.450,-89.605,-176.767,11.353,149.471
C04318=1118.601,390.203,-89.566,-176.769,11.351,149.471
C04319=1118.603,389.991,-89.533,-176.771,11.349,149.471
C04320=1118.607,389.779,-89.501,-176.772,11.346,149.471
C04321=1118.610,389.567,-89.469,-176.774,11.344,149.471
C04322=1118.613,389.356,-89.436,-176.775,11.342,149.471
C04323=1118.617,389.143,-89.403,-176.777,11.340,149.471
C04324=1118.619,388.931,-89.371,-176.779,11.337,149.470
C04325=1118.622,388.720,-89.338,-176.781,11.335,149.470
C04326=1118.625,388.508,-89.306,-176.782,11.333,149.470
C04327=1118.629,388.261,-89.268,-176.785,11.330,149.470
C04328=1118.633,388.014,-89.230,-176.787,11.328,149.470
C04329=1118.637,387.767,-89.192,-176.789,11.326,149.470
C04330=1118.640,387.520,-89.154,-176.790,11.323,149.470
C04331=1118.644,387.273,-89.117,-176.793,11.320,149.469
C04332=1118.648,387.025,-89.079,-176.795,11.318,149.469
C04333=1118.652,386.778,-89.041,-176.797,11.316,149.469
C04334=1118.655,386.531,-89.004,-176.799,11.313,149.469
C04335=1118.658,386.284,-88.966,-176.801,11.311,149.469
C04336=1118.662,386.037,-88.928,-176.804,11.308,149.469
C04337=1118.666,385.790,-88.889,-176.806,11.306,149.469
C04338=1118.670,385.542,-88.853,-176.808,11.303,149.469
C04339=1118.673,385.295,-88.815,-176.810,11.301,149.469
C04340=1118.677,385.049,-88.777,-176.812,11.299,149.469
C04341=1118.680,384.801,-88.739,-176.814,11.297,149.469
C04342=1118.685,384.554,-88.701,-176.816,11.295,149.469
C04343=1118.688,384.307,-88.664,-176.818,11.293,149.469
C04344=1118.692,384.060,-88.626,-176.820,11.291,149.469
C04345=1118.695,383.813,-88.588,-176.823,11.288,149.469
C04346=1118.699,383.566,-88.551,-176.825,11.285,149.469
C04347=1118.703,383.319,-88.514,-176.827,11.283,149.469
C04348=1118.706,383.072,-88.476,-176.831,11.281,149.469
C04349=1118.711,382.825,-88.438,-176.834,11.278,149.469
C04350=1118.714,382.577,-88.400,-176.837,11.276,149.469
C04351=1118.718,382.330,-88.363,-176.840,11.273,149.469
C04352=1118.721,382.083,-88.325,-176.843,11.270,149.469
C04353=1118.725,381.836,-88.288,-176.845,11.268,149.469
C04354=1118.728,381.589,-88.250,-176.849,11.266,149.470
C04355=1118.732,381.341,-88.213,-176.852,11.263,149.470
C04356=1118.736,381.095,-88.176,-176.855,11.260,149.470
C04357=1118.740,380.847,-88.139,-176.858,11.258,149.470
C04358=1118.744,380.600,-88.101,-176.861,11.255,149.470
C04359=1118.747,380.353,-88.063,-176.864,11.252,149.470
C04360=1118.751,380.106,-88.026,-176.867,11.250,149.470
C04361=1118.755,379.859,-87.989,-176.870,11.247,149.470
C04362=1118.758,379.611,-87.951,-176.873,11.245,149.470
C04363=1118.762,379.365,-87.914,-176.876,11.243,149.471
C04364=1118.765,379.117,-87.877,-176.879,11.240,149.471
C04365=1118.769,378.870,-87.840,-176.882,11.238,149.471
C04366=1118.773,378.623,-87.802,-176.886,11.235,149.471
C04367=1118.777,378.375,-87.765,-176.889,11.233,149.471
C04368=1118.781,378.129,-87.727,-176.892,11.230,149.471
C04369=1118.785,377.882,-87.690,-176.895,11.227,149.471
C04370=1118.788,377.634,-87.653,-176.898,11.225,149.472
C04371=1118.792,377.387,-87.616,-176.901,11.223,149.472
C04372=1118.796,377.140,-87.579,-176.904,11.220,149.472
C04373=1118.799,376.893,-87.541,-176.907,11.218,149.472
C04374=1118.803,376.645,-87.504,-176.910,11.215,149.472
C04375=1118.806,376.433,-87.472,-176.913,11.213,149.472
C04376=1118.810,376.221,-87.441,-176.916,11.211,149.473
C04377=1118.813,376.009,-87.409,-176.918,11.209,149.473
C04378=1118.816,375.797,-87.377,-176.921,11.207,149.473
C04379=1118.819,375.586,-87.345,-176.924,11.205,149.473
C04380=1118.822,375.373,-87.314,-176.927,11.203,149.473
C04381=1118.826,375.161,-87.281,-176.929,11.201,149.473
C04382=1118.829,374.950,-87.249,-176.932,11.198,149.473
C04383=1118.833,374.702,-87.213,-176.935,11.196,149.474
C04384=1118.837,374.454,-87.175,-176.939,11.193,149.474
C04385=1118.840,374.208,-87.139,-176.941,11.191,149.474
C04386=1118.844,373.960,-87.102,-176.945,11.189,149.474
C04387=1118.847,373.713,-87.064,-176.948,11.186,149.474
C04388=1118.851,373.466,-87.027,-176.951,11.184,149.475
C04389=1118.856,373.219,-86.991,-176.955,11.181,149.475
C04390=1118.859,372.972,-86.954,-176.958,11.179,149.475
C04391=1118.862,372.724,-86.917,-176.961,11.177,149.475
C04392=1118.866,372.477,-86.880,-176.964,11.174,149.475
C04393=1118.871,372.230,-86.843,-176.968,11.172,149.476
C04394=1118.874,371.983,-86.807,-176.970,11.170,149.476
C04395=1118.877,371.735,-86.770,-176.974,11.167,149.476
C04396=1118.882,371.488,-86.733,-176.977,11.165,149.476
C04397=1118.886,371.240,-86.696,-176.980,11.162,149.476
C04398=1118.889,370.994,-86.660,-176.984,11.160,149.477
C04399=1118.893,370.746,-86.623,-176.987,11.157,149.477
C04400=1118.897,370.498,-86.586,-176.990,11.155,149.477
C04401=1118.900,370.252,-86.550,-176.994,11.153,149.477
C04402=1118.904,370.004,-86.513,-176.997,11.150,149.478
C04403=1118.908,369.757,-86.476,-177.000,11.148,149.478
C04404=1118.911,369.510,-86.440,-177.003,11.146,149.478
C04405=1118.915,369.262,-86.402,-177.006,11.143,149.478
C04406=1118.919,369.015,-86.365,-177.009,11.141,149.478
C04407=1118.922,368.768,-86.329,-177.013,11.139,149.479
C04408=1118.927,368.521,-86.293,-177.016,11.136,149.479
C04409=1118.931,368.273,-86.256,-177.020,11.134,149.479
C04410=1118.934,368.026,-86.220,-177.023,11.131,149.479
C04411=1118.938,367.779,-86.183,-177.026,11.129,149.480
C04412=1118.941,367.532,-86.146,-177.030,11.126,149.480
C04413=1118.945,367.284,-86.110,-177.033,11.124,149.480
C04414=1118.950,367.037,-86.073,-177.036,11.121,149.480
C04415=1118.953,366.790,-86.037,-177.040,11.119,149.481
C04416=1118.957,366.543,-86.000,-177.043,11.117,149.481
C04417=1118.961,366.295,-85.965,-177.046,11.115,149.481
C04418=1118.965,366.048,-85.928,-177.049,11.113,149.481
C04419=1118.968,365.801,-85.892,-177.052,11.110,149.482
C04420=1118.973,365.553,-85.856,-177.056,11.108,149.482
C04421=1118.975,365.306,-85.819,-177.059,11.106,149.482
C04422=1118.979,365.058,-85.782,-177.063,11.103,149.482
C04423=1118.983,364.811,-85.747,-177.066,11.101,149.483
C04424=1118.987,364.564,-85.710,-177.069,11.098,149.483
C04425=1118.991,364.317,-85.673,-177.073,11.096,149.483
C04426=1118.995,364.069,-85.637,-177.076,11.093,149.483
C04427=1118.998,363.822,-85.601,-177.080,11.091,149.484
C04428=1119.003,363.574,-85.565,-177.083,11.089,149.484
C04429=1119.006,363.328,-85.529,-177.086,11.086,149.484
C04430=1119.010,363.080,-85.492,-177.090,11.084,149.484
C04431=1119.013,362.867,-85.462,-177.092,11.082,149.484
C04432=1119.016,362.655,-85.431,-177.096,11.079,149.485
C04433=1119.020,362.443,-85.400,-177.098,11.078,149.485
C04434=1119.023,362.231,-85.368,-177.101,11.076,149.485
C04435=1119.026,362.020,-85.337,-177.104,11.074,149.485
C04436=1119.029,361.807,-85.306,-177.107,11.072,149.486
C04437=1119.032,361.595,-85.275,-177.110,11.069,149.486
C04438=1119.035,361.383,-85.244,-177.113,11.067,149.486
C04439=1119.039,361.135,-85.209,-177.116,11.065,149.486
C04440=1119.043,360.887,-85.172,-177.120,11.063,149.487
C04441=1119.047,360.640,-85.136,-177.123,11.060,149.487
C04442=1119.050,360.393,-85.101,-177.126,11.058,149.487
C04443=1119.055,360.146,-85.065,-177.130,11.056,149.487
C04444=1119.059,359.899,-85.029,-177.133,11.053,149.488
C04445=1119.063,359.651,-84.993,-177.136,11.051,149.488
C04446=1119.067,359.404,-84.957,-177.140,11.048,149.488
C04447=1119.070,359.157,-84.921,-177.143,11.046,149.488
C04448=1119.074,358.909,-84.885,-177.147,11.044,149.489
C04449=1119.078,358.662,-84.850,-177.150,11.041,149.489
C04450=1119.082,358.414,-84.813,-177.153,11.039,149.489
C04451=1119.085,358.167,-84.777,-177.157,11.036,149.489
C04452=1119.089,357.920,-84.742,-177.160,11.034,149.490
C04453=1119.093,357.672,-84.706,-177.164,11.032,149.490
C04454=1119.097,357.424,-84.670,-177.167,11.029,149.490
C04455=1119.101,357.177,-84.634,-177.170,11.027,149.490
C04456=1119.104,356.930,-84.598,-177.174,11.024,149.491
C04457=1119.108,356.682,-84.563,-177.177,11.022,149.491
C04458=1119.112,356.436,-84.527,-177.181,11.020,149.491
C04459=1119.116,356.188,-84.491,-177.185,11.017,149.491
C04460=1119.120,355.940,-84.456,-177.188,11.014,149.492
C04461=1119.124,355.693,-84.420,-177.191,11.012,149.492
C04462=1119.127,355.445,-84.385,-177.195,11.009,149.492
C04463=1119.131,355.198,-84.349,-177.198,11.007,149.493
C04464=1119.135,354.950,-84.314,-177.201,11.005,149.493
C04465=1119.139,354.702,-84.277,-177.205,11.002,149.493
C04466=1119.143,354.456,-84.242,-177.208,11.000,149.493
C04467=1119.147,354.208,-84.207,-177.212,10.997,149.494
C04468=1119.151,353.961,-84.171,-177.215,10.995,149.494
C04469=1119.154,353.713,-84.136,-177.218,10.993,149.494
C04470=1119.158,353.466,-84.100,-177.222,10.989,149.494
C04471=1119.162,353.218,-84.064,-177.226,10.987,149.494
C04472=1119.166,352.971,-84.029,-177.229,10.984,149.495
C04473=1119.170,352.724,-83.994,-177.232,10.982,149.495
C04474=1119.173,352.476,-83.958,-177.236,10.980,149.495
C04475=1119.177,352.229,-83.923,-177.239,10.977,149.496
C04476=1119.181,351.981,-83.888,-177.243,10.975,149.496
C04477=1119.185,351.734,-83.853,-177.247,10.972,149.496
C04478=1119.189,351.486,-83.817,-177.250,10.969,149.496
C04479=1119.193,351.239,-83.782,-177.253,10.967,149.496
C04480=1119.196,350.991,-83.746,-177.256,10.964,149.497
C04481=1119.201,350.744,-83.711,-177.260,10.962,149.497
C04482=1119.204,350.496,-83.676,-177.264,10.960,149.497
C04483=1119.208,350.249,-83.640,-177.267,10.956,149.497
C04484=1119.212,350.001,-83.605,-177.271,10.954,149.498
C04485=1119.216,349.754,-83.570,-177.274,10.951,149.498
C04486=1119.220,349.507,-83.535,-177.277,10.949,149.498
C04487=1119.224,349.294,-83.505,-177.281,10.947,149.498
C04488=1119.227,349.082,-83.474,-177.283,10.945,149.498
C04489=1119.229,348.869,-83.444,-177.286,10.943,149.499
C04490=1119.233,348.657,-83.414,-177.289,10.940,149.499
C04491=1119.236,348.445,-83.384,-177.291,10.938,149.499
C04492=1119.240,348.233,-83.354,-177.294,10.936,149.499
C04493=1119.243,348.020,-83.324,-177.297,10.934,149.499
C04494=1119.247,347.808,-83.294,-177.300,10.932,149.500
C04495=1119.250,347.561,-83.259,-177.303,10.930,149.500
C04496=1119.254,347.313,-83.223,-177.306,10.927,149.500
C04497=1119.259,347.066,-83.189,-177.309,10.924,149.500
C04498=1119.262,346.818,-83.153,-177.312,10.922,149.500
C04499=1119.266,346.570,-83.119,-177.316,10.920,149.501
C04500=1119.270,346.323,-83.083,-177.319,10.917,149.501
C04501=1119.274,346.075,-83.049,-177.322,10.915,149.501
C04502=1119.277,345.828,-83.014,-177.325,10.912,149.501
C04503=1119.282,345.581,-82.979,-177.328,10.910,149.501
C04504=1119.286,345.333,-82.944,-177.331,10.908,149.502
C04505=1119.290,345.085,-82.909,-177.335,10.905,149.502
C04506=1119.294,344.837,-82.874,-177.338,10.903,149.502
C04507=1119.297,344.590,-82.839,-177.341,10.900,149.502
C04508=1119.302,344.343,-82.805,-177.344,10.898,149.502
C04509=1119.305,344.095,-82.769,-177.347,10.895,149.502
C04510=1119.309,343.847,-82.734,-177.351,10.893,149.503
C04511=1119.313,343.600,-82.701,-177.354,10.890,149.503
C04512=1119.317,343.353,-82.665,-177.357,10.888,149.503
C04513=1119.321,343.105,-82.631,-177.360,10.885,149.503
C04514=1119.325,342.857,-82.596,-177.364,10.882,149.503
C04515=1119.329,342.610,-82.562,-177.367,10.880,149.504
C04516=1119.333,342.363,-82.526,-177.370,10.878,149.504
C04517=1119.337,342.114,-82.491,-177.373,10.876,149.504
C04518=1119.341,341.867,-82.458,-177.376,10.873,149.504
C04519=1119.345,341.619,-82.423,-177.379,10.871,149.504
C04520=1119.349,341.372,-82.388,-177.382,10.868,149.505
C04521=1119.352,341.125,-82.353,-177.386,10.866,149.505
C04522=1119.357,340.877,-82.319,-177.389,10.863,149.505
C04523=1119.361,340.629,-82.284,-177.392,10.861,149.505
C04524=1119.364,340.382,-82.250,-177.395,10.858,149.505
C04525=1119.368,340.134,-82.215,-177.399,10.856,149.506
C04526=1119.373,339.887,-82.180,-177.402,10.853,149.506
C04527=1119.376,339.639,-82.146,-177.405,10.851,149.506
C04528=1119.380,339.392,-82.111,-177.408,10.848,149.506
C04529=1119.384,339.144,-82.077,-177.411,10.845,149.506
C04530=1119.388,338.897,-82.043,-177.415,10.843,149.507
C04531=1119.391,338.649,-82.009,-177.417,10.841,149.507
C04532=1119.396,338.401,-81.974,-177.421,10.839,149.507
C04533=1119.400,338.153,-81.939,-177.424,10.836,149.507
C04534=1119.404,337.906,-81.905,-177.427,10.834,149.507
C04535=1119.408,337.658,-81.871,-177.430,10.831,149.508
C04536=1119.412,337.411,-81.837,-177.434,10.829,149.508
C04537=1119.416,337.163,-81.802,-177.437,10.826,149.508
C04538=1119.419,336.916,-81.768,-177.440,10.823,149.508
C04539=1119.424,336.668,-81.733,-177.443,10.821,149.508
C04540=1119.427,336.420,-81.699,-177.447,10.819,149.509
C04541=1119.432,336.173,-81.665,-177.449,10.816,149.509
C04542=1119.435,335.925,-81.631,-177.453,10.813,149.509
C04543=1119.439,335.712,-81.602,-177.455,10.812,149.509
C04544=1119.442,335.500,-81.572,-177.458,10.810,149.509
C04545=1119.445,335.288,-81.542,-177.461,10.807,149.510
C04546=1119.449,335.075,-81.514,-177.463,10.805,149.510
C04547=1119.452,334.863,-81.484,-177.467,10.803,149.510
C04548=1119.456,334.650,-81.455,-177.469,10.801,149.510
C04549=1119.459,334.438,-81.426,-177.472,10.799,149.510
C04550=1119.462,334.226,-81.396,-177.475,10.796,149.510
C04551=1119.467,333.977,-81.362,-177.478,10.794,149.511
C04552=1119.470,333.730,-81.328,-177.481,10.792,149.511
C04553=1119.474,333.483,-81.294,-177.484,10.789,149.511
C04554=1119.478,333.235,-81.260,-177.487,10.787,149.511
C04555=1119.482,332.987,-81.226,-177.490,10.784,149.511
C04556=1119.486,332.739,-81.192,-177.493,10.782,149.511
C04557=1119.490,332.492,-81.158,-177.496,10.779,149.512
C04558=1119.494,332.244,-81.125,-177.500,10.777,149.512
C04559=1119.498,331.996,-81.090,-177.503,10.774,149.512
C04560=1119.502,331.749,-81.056,-177.506,10.772,149.512
C04561=1119.506,331.501,-81.023,-177.509,10.769,149.512
C04562=1119.509,331.253,-80.988,-177.513,10.767,149.513
C04563=1119.513,331.006,-80.955,-177.516,10.764,149.513
C04564=1119.518,330.758,-80.921,-177.519,10.761,149.513
C04565=1119.521,330.510,-80.887,-177.522,10.759,149.513
C04566=1119.526,330.263,-80.853,-177.525,10.757,149.513
C04567=1119.530,330.015,-80.819,-177.528,10.755,149.514
C04568=1119.534,329.768,-80.785,-177.531,10.752,149.514
C04569=1119.537,329.520,-80.752,-177.534,10.750,149.514
C04570=1119.541,329.273,-80.718,-177.537,10.747,149.514
C04571=1119.545,329.025,-80.685,-177.541,10.744,149.514
C04572=1119.549,328.777,-80.650,-177.544,10.742,149.515
C04573=1119.554,328.529,-80.617,-177.547,10.740,149.515
C04574=1119.557,328.282,-80.583,-177.550,10.737,149.515
C04575=1119.562,328.034,-80.550,-177.554,10.734,149.515
C04576=1119.565,327.786,-80.516,-177.557,10.732,149.515
C04577=1119.570,327.538,-80.482,-177.560,10.729,149.515
C04578=1119.574,327.291,-80.448,-177.563,10.727,149.516
C04579=1119.578,327.044,-80.415,-177.566,10.725,149.516
C04580=1119.581,326.795,-80.381,-177.569,10.722,149.516
C04581=1119.585,326.547,-80.348,-177.572,10.720,149.516
C04582=1119.589,326.300,-80.314,-177.575,10.717,149.516
C04583=1119.593,326.053,-80.281,-177.578,10.714,149.517
C04584=1119.597,325.805,-80.248,-177.582,10.712,149.517
C04585=1119.601,325.557,-80.213,-177.585,10.710,149.517
C04586=1119.605,325.309,-80.180,-177.588,10.707,149.517
C04587=1119.610,325.061,-80.147,-177.591,10.704,149.517
C04588=1119.614,324.813,-80.113,-177.594,10.702,149.518
C04589=1119.618,324.566,-80.079,-177.597,10.699,149.518
C04590=1119.621,324.318,-80.046,-177.601,10.697,149.518
C04591=1119.625,324.070,-80.013,-177.604,10.694,149.518
C04592=1119.629,323.822,-79.980,-177.607,10.691,149.518
C04593=1119.633,323.575,-79.946,-177.610,10.690,149.519
C04594=1119.637,323.328,-79.913,-177.613,10.687,149.519
C04595=1119.642,323.080,-79.879,-177.616,10.685,149.519
C04596=1119.645,322.831,-79.846,-177.619,10.682,149.519
C04597=1119.649,322.584,-79.813,-177.623,10.680,149.519
C04598=1119.653,322.336,-79.780,-177.625,10.677,149.519
C04599=1119.656,322.123,-79.751,-177.628,10.675,149.520
C04600=1119.660,321.911,-79.723,-177.631,10.672,149.520
C04601=1119.664,321.698,-79.694,-177.633,10.670,149.520
C04602=1119.667,321.486,-79.666,-177.637,10.668,149.520
C04603=1119.670,321.273,-79.637,-177.639,10.666,149.520
C04604=1119.673,321.061,-79.609,-177.642,10.664,149.520
C04605=1119.677,320.848,-79.580,-177.645,10.662,149.520
C04606=1119.680,320.635,-79.551,-177.647,10.660,149.521
C04607=1119.685,320.388,-79.518,-177.650,10.657,149.521
C04608=1119.688,320.140,-79.485,-177.654,10.655,149.521
C04609=1119.692,319.892,-79.452,-177.657,10.652,149.521
C04610=1119.696,319.645,-79.419,-177.660,10.650,149.521
C04611=1119.700,319.397,-79.386,-177.663,10.647,149.522
C04612=1119.705,319.149,-79.353,-177.666,10.644,149.522
C04613=1119.709,318.901,-79.320,-177.669,10.643,149.522
C04614=1119.713,318.653,-79.287,-177.672,10.640,149.522
C04615=1119.717,318.406,-79.255,-177.675,10.637,149.522
C04616=1119.720,318.157,-79.221,-177.678,10.635,149.523
C04617=1119.724,317.910,-79.188,-177.681,10.632,149.523
C04618=1119.728,317.662,-79.155,-177.685,10.630,149.523
C04619=1119.732,317.414,-79.122,-177.688,10.627,149.523
C04620=1119.736,317.167,-79.089,-177.691,10.625,149.523
C04621=1119.740,316.918,-79.057,-177.694,10.622,149.523
C04622=1119.744,316.671,-79.023,-177.697,10.619,149.524
C04623=1119.749,316.423,-78.990,-177.700,10.617,149.524
C04624=1119.752,316.176,-78.958,-177.704,10.614,149.524
C04625=1119.756,315.927,-78.925,-177.706,10.612,149.524
C04626=1119.761,315.679,-78.892,-177.709,10.610,149.524
C04627=1119.765,315.432,-78.859,-177.712,10.607,149.524
C04628=1119.768,315.184,-78.826,-177.716,10.605,149.525
C04629=1119.773,314.936,-78.794,-177.719,10.602,149.525
C04630=1119.777,314.688,-78.761,-177.722,10.600,149.525
C04631=1119.780,314.441,-78.728,-177.725,10.597,149.525
C04632=1119.785,314.192,-78.696,-177.728,10.594,149.525
C04633=1119.789,313.945,-78.663,-177.731,10.592,149.526
C04634=1119.793,313.698,-78.630,-177.735,10.589,149.526
C04635=1119.797,313.450,-78.598,-177.738,10.587,149.526
C04636=1119.801,313.202,-78.565,-177.741,10.584,149.526
C04637=1119.805,312.954,-78.533,-177.743,10.582,149.526
C04638=1119.809,312.706,-78.500,-177.747,10.580,149.527
C04639=1119.814,312.458,-78.467,-177.750,10.577,149.527
C04640=1119.817,312.210,-78.435,-177.753,10.575,149.527
C04641=1119.821,311.963,-78.402,-177.756,10.572,149.527
C04642=1119.825,311.715,-78.370,-177.759,10.569,149.527
C04643=1119.829,311.467,-78.337,-177.763,10.567,149.527
C04644=1119.833,311.219,-78.304,-177.765,10.564,149.528
C04645=1119.837,310.971,-78.272,-177.769,10.562,149.528
C04646=1119.842,310.723,-78.240,-177.772,10.559,149.528
C04647=1119.846,310.475,-78.208,-177.775,10.557,149.528
C04648=1119.850,310.228,-78.175,-177.778,10.554,149.528
C04649=1119.853,309.980,-78.143,-177.781,10.552,149.529
C04650=1119.858,309.732,-78.110,-177.784,10.550,149.529
C04651=1119.861,309.484,-78.078,-177.787,10.547,149.529
C04652=1119.866,309.236,-78.045,-177.790,10.544,149.529
C04653=1119.870,308.989,-78.013,-177.793,10.542,149.529
C04654=1119.874,308.740,-77.981,-177.797,10.539,149.529
C04655=1119.877,308.527,-77.953,-177.799,10.537,149.530
C04656=1119.881,308.315,-77.925,-177.802,10.535,149.530
C04657=1119.884,308.102,-77.897,-177.804,10.533,149.530
C04658=1119.888,307.889,-77.870,-177.807,10.530,149.530
C04659=1119.891,307.676,-77.842,-177.810,10.528,149.530
C04660=1119.895,307.464,-77.814,-177.812,10.526,149.530
C04661=1119.898,307.251,-77.786,-177.815,10.524,149.530
C04662=1119.902,307.038,-77.759,-177.818,10.522,149.531
C04663=1119.906,306.790,-77.727,-177.821,10.519,149.531
C04664=1119.910,306.542,-77.695,-177.824,10.517,149.531
C04665=1119.914,306.295,-77.662,-177.827,10.514,149.531
C04666=1119.919,306.047,-77.630,-177.831,10.512,149.531
C04667=1119.922,305.799,-77.598,-177.833,10.509,149.531
C04668=1119.926,305.551,-77.566,-177.836,10.507,149.532
C04669=1119.931,305.303,-77.534,-177.839,10.504,149.532
C04670=1119.935,305.055,-77.502,-177.842,10.502,149.532
C04671=1119.939,304.807,-77.471,-177.846,10.500,149.532
C04672=1119.943,304.559,-77.437,-177.849,10.497,149.532
C04673=1119.946,304.311,-77.406,-177.852,10.494,149.533
C04674=1119.951,304.064,-77.374,-177.855,10.492,149.533
C04675=1119.955,303.816,-77.342,-177.858,10.489,149.533
C04676=1119.959,303.568,-77.310,-177.861,10.486,149.533
C04677=1119.963,303.320,-77.278,-177.865,10.484,149.533
C04678=1119.968,303.072,-77.246,-177.867,10.481,149.533
C04679=1119.971,302.824,-77.214,-177.870,10.480,149.534
C04680=1119.975,302.576,-77.182,-177.873,10.477,149.534
C04681=1119.980,302.328,-77.150,-177.876,10.474,149.534
C04682=1119.984,302.080,-77.118,-177.879,10.472,149.534
C04683=1119.987,301.832,-77.086,-177.883,10.469,149.534
C04684=1119.992,301.585,-77.055,-177.886,10.466,149.535
C04685=1119.996,301.336,-77.023,-177.889,10.464,149.535
C04686=1120.000,301.088,-76.991,-177.892,10.461,149.535
C04687=1120.005,300.840,-76.960,-177.895,10.459,149.535
C04688=1120.008,300.592,-76.928,-177.898,10.456,149.535
C04689=1120.013,300.344,-76.896,-177.901,10.454,149.536
C04690=1120.017,300.097,-76.864,-177.904,10.452,149.536
C04691=1120.021,299.849,-76.832,-177.907,10.449,149.536
C04692=1120.024,299.601,-76.800,-177.910,10.446,149.536
C04693=1120.029,299.353,-76.770,-177.913,10.444,149.536
C04694=1120.033,299.105,-76.738,-177.916,10.441,149.536
C04695=1120.038,298.857,-76.706,-177.920,10.439,149.537
C04696=1120.042,298.609,-76.674,-177.923,10.436,149.537
C04697=1120.045,298.361,-76.642,-177.926,10.434,149.537
C04698=1120.050,298.113,-76.611,-177.929,10.431,149.537
C04699=1120.054,297.865,-76.579,-177.932,10.428,149.537
C04700=1120.058,297.618,-76.548,-177.935,10.426,149.537
C04701=1120.062,297.369,-76.517,-177.938,10.424,149.538
C04702=1120.066,297.121,-76.485,-177.941,10.421,149.538
C04703=1120.070,296.874,-76.454,-177.944,10.419,149.538
C04704=1120.075,296.625,-76.422,-177.947,10.416,149.538
C04705=1120.079,296.377,-76.390,-177.950,10.414,149.538
C04706=1120.083,296.129,-76.358,-177.953,10.411,149.538
C04707=1120.087,295.881,-76.327,-177.957,10.408,149.539
C04708=1120.091,295.633,-76.296,-177.960,10.406,149.539
C04709=1120.095,295.385,-76.264,-177.963,10.403,149.539
C04710=1120.099,295.137,-76.233,-177.966,10.400,149.539
C04711=1120.103,294.925,-76.206,-177.968,10.398,149.539
C04712=1120.106,294.711,-76.180,-177.971,10.397,149.540
C04713=1120.109,294.499,-76.153,-177.974,10.394,149.540
C04714=1120.113,294.286,-76.126,-177.976,10.392,149.540
C04715=1120.116,294.072,-76.099,-177.979,10.390,149.540
C04716=1120.120,293.859,-76.072,-177.982,10.388,149.540
C04717=1120.123,293.647,-76.045,-177.984,10.386,149.540
C04718=1120.127,293.434,-76.019,-177.986,10.384,149.540
C04719=1120.131,293.186,-75.987,-177.990,10.381,149.541
C04720=1120.136,292.938,-75.956,-177.993,10.378,149.541
C04721=1120.139,292.690,-75.924,-177.996,10.376,149.541
C04722=1120.144,292.442,-75.894,-177.999,10.373,149.541
C04723=1120.148,292.194,-75.862,-178.002,10.371,149.541
C04724=1120.152,291.946,-75.831,-178.005,10.368,149.541
C04725=1120.156,291.697,-75.800,-178.008,10.366,149.542
C04726=1120.160,291.450,-75.769,-178.011,10.363,149.542
C04727=1120.164,291.202,-75.738,-178.014,10.361,149.542
C04728=1120.168,290.954,-75.707,-178.017,10.358,149.542
C04729=1120.172,290.706,-75.675,-178.020,10.356,149.542
C04730=1120.177,290.458,-75.645,-178.023,10.353,149.543
C04731=1120.181,290.209,-75.613,-178.026,10.350,149.543
C04732=1120.185,289.962,-75.582,-178.030,10.348,149.543
C04733=1120.188,289.713,-75.551,-178.033,10.345,149.543
C04734=1120.193,289.466,-75.521,-178.036,10.343,149.543
C04735=1120.198,289.218,-75.490,-178.039,10.340,149.543
C04736=1120.201,288.970,-75.458,-178.042,10.338,149.544
C04737=1120.206,288.722,-75.427,-178.044,10.336,149.544
C04738=1120.209,288.473,-75.397,-178.047,10.333,149.544
C04739=1120.214,288.225,-75.366,-178.051,10.330,149.544
C04740=1120.218,287.977,-75.335,-178.054,10.328,149.544
C04741=1120.222,287.729,-75.303,-178.057,10.325,149.545
C04742=1120.226,287.482,-75.273,-178.060,10.323,149.545
C04743=1120.230,287.233,-75.242,-178.063,10.320,149.545
C04744=1120.235,286.985,-75.211,-178.066,10.317,149.545
C04745=1120.239,286.737,-75.181,-178.070,10.315,149.545
C04746=1120.243,286.489,-75.150,-178.072,10.313,149.545
C04747=1120.247,286.241,-75.119,-178.075,10.310,149.545
C04748=1120.252,285.993,-75.089,-178.078,10.308,149.546
C04749=1120.255,285.744,-75.058,-178.081,10.305,149.546
C04750=1120.260,285.496,-75.027,-178.084,10.303,149.546
C04751=1120.264,285.248,-74.996,-178.087,10.300,149.546
C04752=1120.268,285.000,-74.966,-178.091,10.297,149.546
C04753=1120.272,284.752,-74.935,-178.094,10.295,149.547
C04754=1120.277,284.504,-74.904,-178.097,10.292,149.547
C04755=1120.280,284.256,-74.874,-178.100,10.289,149.547
C04756=1120.285,284.008,-74.843,-178.102,10.287,149.547
C04757=1120.289,283.760,-74.813,-178.106,10.285,149.547
C04758=1120.293,283.512,-74.782,-178.108,10.282,149.547
C04759=1120.297,283.264,-74.751,-178.112,10.280,149.548
C04760=1120.301,283.016,-74.721,-178.115,10.277,149.548
C04761=1120.306,282.768,-74.690,-178.118,10.274,149.548
C04762=1120.309,282.520,-74.660,-178.121,10.272,149.548
C04763=1120.314,282.272,-74.629,-178.124,10.269,149.548
C04764=1120.318,282.023,-74.599,-178.127,10.267,149.549
C04765=1120.322,281.776,-74.569,-178.130,10.265,149.549
C04766=1120.326,281.527,-74.537,-178.133,10.262,149.549
C04767=1120.330,281.314,-74.512,-178.136,10.260,149.549
C04768=1120.333,281.101,-74.486,-178.139,10.257,149.549
C04769=1120.337,280.888,-74.459,-178.142,10.255,149.549
C04770=1120.340,280.675,-74.433,-178.144,10.252,149.550
C04771=1120.344,280.462,-74.407,-178.147,10.250,149.550
C04772=1120.348,280.249,-74.382,-178.150,10.248,149.550
C04773=1120.352,280.036,-74.355,-178.153,10.245,149.550
C04774=1120.355,279.823,-74.329,-178.155,10.243,149.550
C04775=1120.360,279.575,-74.298,-178.159,10.241,149.550
C04776=1120.364,279.327,-74.269,-178.162,10.238,149.551
C04777=1120.367,279.078,-74.238,-178.166,10.235,149.551
C04778=1120.372,278.830,-74.208,-178.169,10.232,149.551
C04779=1120.376,278.582,-74.178,-178.172,10.230,149.551
C04780=1120.380,278.334,-74.147,-178.175,10.227,149.551
C04781=1120.385,278.086,-74.118,-178.178,10.224,149.551
C04782=1120.388,277.838,-74.088,-178.181,10.222,149.552
C04783=1120.392,277.590,-74.057,-178.184,10.219,149.552
C04784=1120.397,277.341,-74.027,-178.187,10.216,149.552
C04785=1120.401,277.093,-73.996,-178.190,10.214,149.552
C04786=1120.405,276.845,-73.967,-178.193,10.211,149.552
C04787=1120.409,276.597,-73.937,-178.196,10.208,149.552
C04788=1120.414,276.349,-73.907,-178.200,10.205,149.553
C04789=1120.418,276.101,-73.876,-178.203,10.202,149.553
C04790=1120.422,275.852,-73.847,-178.206,10.200,149.553
C04791=1120.426,275.605,-73.817,-178.209,10.197,149.553
C04792=1120.431,275.356,-73.787,-178.212,10.194,149.553
C04793=1120.434,275.108,-73.756,-178.215,10.192,149.553
C04794=1120.439,274.860,-73.727,-178.218,10.189,149.553
C04795=1120.443,274.612,-73.697,-178.221,10.186,149.553
C04796=1120.447,274.364,-73.667,-178.224,10.183,149.554
C04797=1120.452,274.116,-73.637,-178.226,10.181,149.554
C04798=1120.455,273.868,-73.607,-178.230,10.179,149.554
C04799=1120.460,273.619,-73.577,-178.233,10.176,149.554
C04800=1120.464,273.370,-73.547,-178.236,10.173,149.554
C04801=1120.468,273.123,-73.517,-178.239,10.171,149.554
C04802=1120.472,272.875,-73.488,-178.242,10.168,149.554
C04803=1120.476,272.626,-73.458,-178.244,10.165,149.554
C04804=1120.481,272.378,-73.427,-178.247,10.162,149.555
C04805=1120.485,272.130,-73.398,-178.250,10.160,149.555
C04806=1120.489,271.882,-73.369,-178.253,10.157,149.555
C04807=1120.493,271.634,-73.339,-178.256,10.155,149.555
C04808=1120.497,271.386,-73.309,-178.259,10.153,149.555
C04809=1120.501,271.138,-73.279,-178.262,10.150,149.555
C04810=1120.506,270.889,-73.249,-178.265,10.147,149.555
C04811=1120.510,270.641,-73.220,-178.268,10.144,149.555
C04812=1120.515,270.392,-73.191,-178.271,10.141,149.556
C04813=1120.519,270.144,-73.161,-178.273,10.140,149.556
C04814=1120.523,269.897,-73.131,-178.276,10.137,149.556
C04815=1120.527,269.648,-73.101,-178.279,10.134,149.556
C04816=1120.531,269.400,-73.072,-178.282,10.131,149.556
C04817=1120.535,269.152,-73.043,-178.284,10.129,149.556
C04818=1120.539,268.903,-73.013,-178.287,10.126,149.556
C04819=1120.544,268.655,-72.984,-178.290,10.124,149.556
C04820=1120.549,268.407,-72.954,-178.292,10.122,149.556
C04821=1120.553,268.158,-72.924,-178.295,10.119,149.557
C04822=1120.557,267.910,-72.895,-178.298,10.116,149.557
C04823=1120.560,267.697,-72.869,-178.300,10.114,149.557
C04824=1120.564,267.485,-72.844,-178.302,10.112,149.557
C04825=1120.568,267.271,-72.819,-178.305,10.110,149.557
C04826=1120.571,267.058,-72.794,-178.307,10.108,149.557
C04827=1120.575,266.844,-72.768,-178.309,10.106,149.557
C04828=1120.578,266.632,-72.743,-178.312,10.104,149.557
C04829=1120.582,266.419,-72.718,-178.314,10.101,149.557
C04830=1120.586,266.205,-72.693,-178.316,10.099,149.557
C04831=1120.590,265.957,-72.663,-178.319,10.097,149.557
C04832=1120.594,265.709,-72.634,-178.322,10.094,149.557
C04833=1120.599,265.461,-72.604,-178.324,10.092,149.558
C04834=1120.603,265.212,-72.575,-178.327,10.089,149.558
C04835=1120.607,264.963,-72.546,-178.329,10.087,149.558
C04836=1120.611,264.715,-72.517,-178.332,10.085,149.558
C04837=1120.616,264.467,-72.487,-178.334,10.083,149.558
C04838=1120.620,264.219,-72.458,-178.338,10.080,149.558
C04839=1120.625,263.971,-72.429,-178.341,10.077,149.558
C04840=1120.629,263.723,-72.399,-178.345,10.074,149.559
C04841=1120.632,263.475,-72.370,-178.348,10.071,149.559
C04842=1120.637,263.226,-72.341,-178.352,10.068,149.559
C04843=1120.641,262.978,-72.312,-178.355,10.065,149.559
C04844=1120.646,262.730,-72.283,-178.358,10.062,149.559
C04845=1120.650,262.482,-72.253,-178.362,10.059,149.560
C04846=1120.654,262.233,-72.225,-178.365,10.056,149.560
C04847=1120.658,261.985,-72.195,-178.369,10.053,149.560
C04848=1120.662,261.737,-72.166,-178.372,10.050,149.560
C04849=1120.666,261.488,-72.138,-178.375,10.048,149.560
C04850=1120.671,261.240,-72.109,-178.379,10.044,149.560
C04851=1120.675,260.992,-72.079,-178.382,10.041,149.560
C04852=1120.680,260.743,-72.050,-178.385,10.039,149.561
C04853=1120.683,260.495,-72.022,-178.388,10.036,149.561
C04854=1120.687,260.247,-71.992,-178.391,10.033,149.561
C04855=1120.693,259.999,-71.964,-178.394,10.030,149.561
C04856=1120.697,259.750,-71.934,-178.397,10.027,149.561
C04857=1120.700,259.502,-71.906,-178.400,10.024,149.561
C04858=1120.705,259.254,-71.877,-178.403,10.021,149.561
C04859=1120.710,259.005,-71.848,-178.406,10.019,149.561
C04860=1120.714,258.757,-71.819,-178.410,10.015,149.562
C04861=1120.717,258.509,-71.790,-178.413,10.012,149.562
C04862=1120.722,258.260,-71.761,-178.416,10.010,149.562
C04863=1120.727,258.013,-71.732,-178.418,10.007,149.562
C04864=1120.730,257.764,-71.704,-178.421,10.004,149.562
C04865=1120.735,257.515,-71.675,-178.424,10.001,149.562
C04866=1120.740,257.268,-71.646,-178.427,9.998,149.562
C04867=1120.743,257.019,-71.618,-178.430,9.996,149.562
C04868=1120.748,256.771,-71.589,-178.433,9.993,149.562
C04869=1120.752,256.522,-71.560,-178.436,9.990,149.562
C04870=1120.756,256.275,-71.531,-178.438,9.987,149.562
C04871=1120.761,256.026,-71.503,-178.441,9.984,149.562
C04872=1120.764,255.777,-71.474,-178.442,9.982,149.562
C04873=1120.769,255.530,-71.445,-178.443,9.981,149.562
C04874=1120.774,255.281,-71.417,-178.443,9.980,149.562
C04875=1120.777,255.032,-71.389,-178.445,9.978,149.562
C04876=1120.782,254.785,-71.359,-178.446,9.976,149.562
C04877=1120.786,254.536,-71.331,-178.447,9.975,149.562
C04878=1120.790,254.287,-71.303,-178.448,9.973,149.561
C04879=1120.796,253.963,-71.265,-178.450,9.971,149.562
C04880=1120.801,253.639,-71.228,-178.453,9.968,149.562
C04881=1120.807,253.315,-71.190,-178.455,9.966,149.562
C04882=1120.813,252.990,-71.153,-178.458,9.963,149.562
C04883=1120.817,252.743,-71.125,-178.461,9.960,149.562
C04884=1120.822,252.494,-71.096,-178.463,9.958,149.562
C04885=1120.825,252.246,-71.068,-178.466,9.956,149.562
C04886=1120.830,251.997,-71.039,-178.469,9.954,149.562
C04887=1120.834,251.750,-71.011,-178.472,9.951,149.563
C04888=1120.839,251.501,-70.982,-178.475,9.949,149.563
C04889=1120.843,251.253,-70.954,-178.479,9.945,149.563
C04890=1120.847,251.004,-70.926,-178.482,9.943,149.563
C04891=1120.851,250.755,-70.897,-178.486,9.940,149.564
C04892=1120.856,250.508,-70.868,-178.490,9.937,149.564
C04893=1120.860,250.259,-70.840,-178.494,9.933,149.564
C04894=1120.865,250.011,-70.812,-178.498,9.930,149.564
C04895=1120.871,249.660,-70.772,-178.505,9.925,149.565
C04896=1120.877,249.309,-70.732,-178.511,9.920,149.565
C04897=1120.883,248.958,-70.693,-178.517,9.915,149.566
C04898=1120.889,248.608,-70.652,-178.524,9.909,149.566
C04899=1120.893,248.359,-70.624,-178.529,9.905,149.567
C04900=1120.897,248.111,-70.596,-178.534,9.901,149.567
C04901=1120.902,247.862,-70.568,-178.540,9.896,149.567
C04902=1120.906,247.614,-70.540,-178.545,9.892,149.568
C04903=1120.910,247.366,-70.512,-178.549,9.888,149.568
C04904=1120.915,247.117,-70.484,-178.551,9.886,149.568
C04905=1120.919,246.868,-70.456,-178.552,9.883,149.567
C04906=1120.923,246.620,-70.428,-178.554,9.881,149.567
C04907=1120.927,246.372,-70.400,-178.556,9.878,149.567
C04908=1120.932,246.124,-70.372,-178.558,9.876,149.567
C04909=1120.936,245.876,-70.344,-178.560,9.873,149.567
C04910=1120.940,245.627,-70.316,-178.561,9.871,149.567
C04911=1120.945,245.379,-70.289,-178.563,9.869,149.567
C04912=1120.949,245.130,-70.260,-178.565,9.866,149.567
C04913=1120.954,244.882,-70.232,-178.567,9.864,149.567
C04914=1120.957,244.633,-70.204,-178.569,9.862,149.567
C04915=1120.962,244.385,-70.177,-178.571,9.859,149.567
C04916=1120.966,244.136,-70.149,-178.573,9.857,149.567
C04917=1120.971,243.888,-70.120,-178.575,9.855,149.567
C04918=1120.975,243.640,-70.093,-178.577,9.853,149.567
C04919=1120.979,243.391,-70.065,-178.580,9.850,149.567
C04920=1120.984,243.143,-70.037,-178.581,9.847,149.566
C04921=1120.987,242.895,-70.009,-178.583,9.845,149.566
C04922=1120.993,242.646,-69.982,-178.586,9.843,149.567
C04923=1120.997,242.398,-69.954,-178.588,9.841,149.566
C04924=1121.001,242.149,-69.926,-178.590,9.837,149.566
C04925=1121.005,241.901,-69.899,-178.592,9.835,149.567
C04926=1121.009,241.652,-69.870,-178.594,9.833,149.566
C04927=1121.014,241.404,-69.843,-178.597,9.830,149.567
C04928=1121.018,241.156,-69.816,-178.599,9.828,149.567
C04929=1121.023,240.907,-69.787,-178.601,9.826,149.567
C04930=1121.027,240.659,-69.760,-178.604,9.823,149.567
C04931=1121.030,240.445,-69.736,-178.606,9.821,149.567
C04932=1121.034,240.232,-69.712,-178.608,9.819,149.567
C04933=1121.038,240.019,-69.689,-178.610,9.817,149.567
C04934=1121.042,239.805,-69.664,-178.612,9.814,149.567
C04935=1121.046,239.592,-69.641,-178.615,9.812,149.567
C04936=1121.049,239.378,-69.617,-178.617,9.810,149.567
C04937=1121.053,239.165,-69.593,-178.619,9.808,149.567
C04938=1121.057,238.952,-69.569,-178.621,9.806,149.567
C04939=1121.061,238.702,-69.542,-178.623,9.804,149.567
C04940=1121.065,238.455,-69.514,-178.626,9.801,149.567
C04941=1121.070,238.206,-69.487,-178.628,9.799,149.567
C04942=1121.074,237.957,-69.460,-178.631,9.796,149.567
C04943=1121.078,237.709,-69.432,-178.634,9.793,149.567
C04944=1121.083,237.460,-69.405,-178.636,9.791,149.568
C04945=1121.087,237.212,-69.377,-178.639,9.788,149.568
C04946=1121.091,236.963,-69.350,-178.642,9.785,149.568
C04947=1121.096,236.716,-69.322,-178.645,9.783,149.568
C04948=1121.100,236.467,-69.295,-178.647,9.781,149.568
C04949=1121.104,236.218,-69.267,-178.650,9.778,149.568
C04950=1121.109,235.970,-69.240,-178.653,9.775,149.568
C04951=1121.114,235.721,-69.213,-178.656,9.772,149.568
C04952=1121.118,235.472,-69.185,-178.659,9.770,149.568
C04953=1121.122,235.224,-69.157,-178.662,9.767,149.568
C04954=1121.127,234.976,-69.130,-178.664,9.764,149.568
C04955=1121.130,234.728,-69.104,-178.667,9.761,149.569
C04956=1121.134,234.479,-69.076,-178.670,9.758,149.569
C04957=1121.139,234.231,-69.049,-178.673,9.756,149.569
C04958=1121.144,233.982,-69.022,-178.676,9.753,149.569
C04959=1121.148,233.734,-68.995,-178.679,9.750,149.569
C04960=1121.152,233.485,-68.966,-178.682,9.747,149.569
C04961=1121.157,233.237,-68.939,-178.685,9.745,149.569
C04962=1121.161,232.988,-68.912,-178.688,9.742,149.569
C04963=1121.165,232.740,-68.886,-178.691,9.738,149.570
C04964=1121.170,232.491,-68.859,-178.694,9.736,149.570
C04965=1121.174,232.242,-68.831,-178.697,9.733,149.570
C04966=1121.178,231.994,-68.804,-178.700,9.730,149.570
C04967=1121.183,231.746,-68.777,-178.704,9.727,149.570
C04968=1121.188,231.497,-68.749,-178.707,9.724,149.570
C04969=1121.191,231.249,-68.723,-178.710,9.721,149.570
C04970=1121.196,231.001,-68.696,-178.713,9.718,149.570
C04971=1121.200,230.751,-68.668,-178.716,9.715,149.570
C04972=1121.205,230.503,-68.641,-178.720,9.711,149.571
C04973=1121.209,230.255,-68.615,-178.723,9.709,149.571
C04974=1121.213,230.006,-68.588,-178.726,9.705,149.571
C04975=1121.218,229.758,-68.561,-178.730,9.701,149.571
C04976=1121.223,229.509,-68.534,-178.732,9.698,149.571
C04977=1121.227,229.261,-68.507,-178.736,9.695,149.571
C04978=1121.231,229.012,-68.480,-178.739,9.692,149.571
C04979=1121.235,228.763,-68.453,-178.742,9.689,149.571
C04980=1121.239,228.515,-68.426,-178.745,9.686,149.571
C04981=1121.244,228.267,-68.399,-178.749,9.682,149.571
C04982=1121.249,228.018,-68.372,-178.751,9.679,149.571
C04983=1121.253,227.769,-68.346,-178.755,9.676,149.572
C04984=1121.257,227.521,-68.319,-178.758,9.673,149.572
C04985=1121.262,227.272,-68.292,-178.761,9.669,149.572
C04986=1121.266,227.024,-68.266,-178.764,9.666,149.572
C04987=1121.270,226.811,-68.243,-178.767,9.663,149.572
C04988=1121.273,226.597,-68.219,-178.770,9.660,149.572
C04989=1121.277,226.383,-68.196,-178.772,9.657,149.572
C04990=1121.281,226.170,-68.174,-178.775,9.655,149.572
C04991=1121.285,225.956,-68.151,-178.777,9.652,149.572
C04992=1121.289,225.743,-68.129,-178.780,9.649,149.572
C04993=1121.292,225.530,-68.105,-178.782,9.646,149.572
C04994=1121.296,225.316,-68.082,-178.784,9.644,149.572
C04995=1121.301,225.067,-68.057,-178.788,9.640,149.572
C04996=1121.305,224.818,-68.029,-178.790,9.637,149.572
C04997=1121.309,224.569,-68.002,-178.793,9.634,149.572
C04998=1121.313,224.321,-67.976,-178.796,9.630,149.572
C04999=1121.318,224.072,-67.949,-178.799,9.627,149.572
C05000=1121.323,223.825,-67.923,-178.802,9.625,149.572
C05001=1121.328,223.576,-67.897,-178.804,9.621,149.572
C05002=1121.332,223.327,-67.870,-178.807,9.618,149.572
C05003=1121.336,223.079,-67.844,-178.810,9.614,149.572
C05004=1121.341,222.830,-67.818,-178.812,9.611,149.571
C05005=1121.344,222.582,-67.791,-178.815,9.608,149.571
C05006=1121.349,222.333,-67.765,-178.817,9.605,149.571
C05007=1121.353,222.085,-67.738,-178.820,9.602,149.571
C05008=1121.358,221.835,-67.712,-178.822,9.599,149.571
C05009=1121.362,221.587,-67.686,-178.825,9.596,149.571
C05010=1121.366,221.338,-67.660,-178.828,9.593,149.571
C05011=1121.371,221.090,-67.633,-178.831,9.589,149.571
C05012=1121.375,220.841,-67.607,-178.833,9.586,149.571
C05013=1121.380,220.593,-67.580,-178.836,9.583,149.571
C05014=1121.384,220.344,-67.554,-178.838,9.580,149.571
C05015=1121.388,220.096,-67.528,-178.840,9.577,149.571
C05016=1121.393,219.847,-67.501,-178.843,9.574,149.571
C05017=1121.398,219.599,-67.475,-178.845,9.571,149.571
C05018=1121.402,219.350,-67.449,-178.847,9.567,149.570
C05019=1121.407,219.101,-67.423,-178.850,9.564,149.570
C05020=1121.411,218.853,-67.397,-178.852,9.561,149.570
C05021=1121.415,218.604,-67.371,-178.855,9.558,149.570
C05022=1121.420,218.355,-67.345,-178.857,9.555,149.570
C05023=1121.424,218.107,-67.318,-178.859,9.552,149.570
C05024=1121.428,217.858,-67.292,-178.861,9.549,149.570
C05025=1121.433,217.610,-67.267,-178.864,9.546,149.570
C05026=1121.438,217.361,-67.240,-178.866,9.543,149.570
C05027=1121.442,217.113,-67.214,-178.868,9.540,149.569
C05028=1121.446,216.864,-67.188,-178.870,9.537,149.569
C05029=1121.450,216.616,-67.162,-178.873,9.534,149.569
C05030=1121.455,216.367,-67.136,-178.874,9.531,149.569
C05031=1121.459,216.118,-67.110,-178.877,9.528,149.569
C05032=1121.464,215.870,-67.084,-178.879,9.526,149.569
C05033=1121.468,215.621,-67.058,-178.881,9.522,149.569
C05034=1121.473,215.372,-67.032,-178.883,9.520,149.569
C05035=1121.477,215.124,-67.006,-178.885,9.517,149.569
C05036=1121.481,214.875,-66.980,-178.887,9.514,149.568
C05037=1121.486,214.627,-66.955,-178.889,9.511,149.568
C05038=1121.490,214.378,-66.928,-178.891,9.509,149.568
C05039=1121.495,214.129,-66.902,-178.893,9.505,149.568
C05040=1121.499,213.881,-66.876,-178.895,9.503,149.568
C05041=1121.503,213.632,-66.850,-178.897,9.500,149.568
C05042=1121.508,213.384,-66.825,-178.899,9.497,149.568
C05043=1121.512,213.170,-66.803,-178.901,9.495,149.568
C05044=1121.516,212.956,-66.781,-178.903,9.493,149.568
C05045=1121.519,212.743,-66.759,-178.905,9.490,149.568
C05046=1121.523,212.529,-66.736,-178.906,9.488,149.567
C05047=1121.527,212.315,-66.714,-178.908,9.485,149.567
C05048=1121.531,212.101,-66.692,-178.910,9.483,149.567
C05049=1121.534,211.887,-66.670,-178.912,9.481,149.567
C05050=1121.539,211.674,-66.647,-178.914,9.478,149.567
C05051=1121.543,211.425,-66.622,-178.917,9.475,149.567
C05052=1121.548,211.177,-66.596,-178.919,9.472,149.567
C05053=1121.552,210.928,-66.570,-178.921,9.470,149.567
C05054=1121.556,210.679,-66.545,-178.924,9.467,149.567
C05055=1121.560,210.430,-66.519,-178.926,9.464,149.567
C05056=1121.565,210.182,-66.493,-178.928,9.462,149.567
C05057=1121.569,209.934,-66.468,-178.931,9.458,149.567
C05058=1121.574,209.685,-66.442,-178.934,9.456,149.567
C05059=1121.578,209.437,-66.417,-178.936,9.453,149.567
C05060=1121.583,209.188,-66.391,-178.938,9.450,149.567
C05061=1121.587,208.938,-66.366,-178.941,9.447,149.567
C05062=1121.592,208.690,-66.340,-178.944,9.444,149.567
C05063=1121.596,208.442,-66.315,-178.947,9.442,149.567
C05064=1121.600,208.193,-66.289,-178.949,9.439,149.567
C05065=1121.605,207.945,-66.264,-178.952,9.437,149.567
C05066=1121.609,207.696,-66.238,-178.954,9.433,149.567
C05067=1121.614,207.447,-66.212,-178.957,9.431,149.567
C05068=1121.619,207.198,-66.187,-178.960,9.428,149.567
C05069=1121.623,206.949,-66.162,-178.962,9.425,149.567
C05070=1121.627,206.701,-66.136,-178.965,9.422,149.568
C05071=1121.632,206.453,-66.110,-178.968,9.419,149.568
C05072=1121.636,206.204,-66.085,-178.971,9.416,149.568
C05073=1121.641,205.954,-66.060,-178.974,9.414,149.568
C05074=1121.646,205.706,-66.034,-178.976,9.410,149.568
C05075=1121.650,205.457,-66.009,-178.979,9.408,149.568
C05076=1121.655,205.209,-65.983,-178.982,9.405,149.568
C05077=1121.659,204.960,-65.958,-178.985,9.402,149.568
C05078=1121.663,204.711,-65.933,-178.988,9.399,149.568
C05079=1121.668,204.463,-65.908,-178.991,9.396,149.568
C05080=1121.672,204.214,-65.883,-178.994,9.394,149.568
C05081=1121.677,203.966,-65.857,-178.997,9.391,149.569
C05082=1121.681,203.716,-65.832,-178.999,9.388,149.569
C05083=1121.686,203.468,-65.807,-179.002,9.385,149.569
C05084=1121.690,203.219,-65.781,-179.006,9.381,149.569
C05085=1121.695,202.971,-65.757,-179.009,9.379,149.569
C05086=1121.699,202.722,-65.731,-179.012,9.376,149.569
C05087=1121.704,202.473,-65.706,-179.014,9.373,149.569
C05088=1121.708,202.225,-65.681,-179.018,9.369,149.569
C05089=1121.712,201.976,-65.656,-179.021,9.367,149.569
C05090=1121.717,201.727,-65.631,-179.024,9.364,149.569
C05091=1121.722,201.478,-65.606,-179.027,9.360,149.570
C05092=1121.726,201.230,-65.581,-179.030,9.358,149.570
C05093=1121.730,200.981,-65.556,-179.033,9.354,149.570
C05094=1121.735,200.733,-65.531,-179.036,9.351,149.570
C05095=1121.740,200.483,-65.506,-179.039,9.348,149.570
C05096=1121.744,200.236,-65.481,-179.043,9.345,149.570
C05097=1121.748,199.986,-65.456,-179.046,9.341,149.570
C05098=1121.753,199.738,-65.430,-179.049,9.339,149.570
C05099=1121.757,199.524,-65.409,-179.052,9.335,149.570
C05100=1121.761,199.309,-65.388,-179.055,9.333,149.571
C05101=1121.765,199.096,-65.367,-179.058,9.330,149.571
C05102=1121.768,198.882,-65.346,-179.060,9.327,149.571
C05103=1121.772,198.668,-65.324,-179.063,9.324,149.571
C05104=1121.776,198.454,-65.303,-179.066,9.321,149.571
C05105=1121.780,198.241,-65.282,-179.069,9.318,149.571
C05106=1121.783,198.027,-65.260,-179.072,9.315,149.571
C05107=1121.789,197.778,-65.235,-179.075,9.312,149.571
C05108=1121.792,197.530,-65.210,-179.078,9.308,149.571
C05109=1121.797,197.281,-65.186,-179.082,9.305,149.571
C05110=1121.802,197.032,-65.161,-179.086,9.301,149.571
C05111=1121.806,196.783,-65.136,-179.088,9.298,149.571
C05112=1121.811,196.535,-65.112,-179.092,9.294,149.571
C05113=1121.815,196.286,-65.087,-179.095,9.291,149.571
C05114=1121.820,196.037,-65.062,-179.097,9.288,149.571
C05115=1121.824,195.789,-65.038,-179.098,9.286,149.571
C05116=1121.829,195.540,-65.013,-179.100,9.283,149.571
C05117=1121.833,195.291,-64.989,-179.102,9.280,149.571
C05118=1121.838,195.042,-64.964,-179.104,9.277,149.571
C05119=1121.842,194.793,-64.940,-179.106,9.275,149.571
C05120=1121.847,194.545,-64.915,-179.107,9.272,149.571
C05121=1121.851,194.296,-64.890,-179.109,9.270,149.570
C05122=1121.856,194.047,-64.865,-179.111,9.267,149.570
C05123=1121.860,193.799,-64.841,-179.113,9.264,149.570
C05124=1121.865,193.550,-64.816,-179.115,9.262,149.570
C05125=1121.869,193.301,-64.792,-179.117,9.259,149.570
C05126=1121.874,193.052,-64.767,-179.119,9.257,149.570
C05127=1121.878,192.803,-64.743,-179.121,9.253,149.570
C05128=1121.882,192.555,-64.719,-179.123,9.251,149.570
C05129=1121.888,192.306,-64.694,-179.124,9.249,149.570
C05130=1121.891,192.057,-64.670,-179.127,9.246,149.569
C05131=1121.896,191.808,-64.645,-179.128,9.243,149.569
C05132=1121.901,191.560,-64.621,-179.131,9.240,149.569
C05133=1121.905,191.312,-64.597,-179.133,9.237,149.569
C05134=1121.910,191.062,-64.572,-179.135,9.235,149.569
C05135=1121.914,190.814,-64.548,-179.137,9.232,149.569
C05136=1121.919,190.565,-64.523,-179.139,9.230,149.569
C05137=1121.923,190.315,-64.499,-179.141,9.226,149.569
C05138=1121.928,190.067,-64.475,-179.143,9.224,149.569
C05139=1121.933,189.818,-64.451,-179.146,9.221,149.569
C05140=1121.937,189.570,-64.427,-179.148,9.218,149.569
C05141=1121.941,189.321,-64.402,-179.150,9.215,149.569
C05142=1121.946,189.072,-64.377,-179.152,9.213,149.569
C05143=1121.951,188.823,-64.353,-179.154,9.210,149.569
C05144=1121.955,188.575,-64.329,-179.156,9.208,149.569
C05145=1121.960,188.325,-64.305,-179.159,9.204,149.568
C05146=1121.964,188.077,-64.281,-179.161,9.201,149.568
C05147=1121.969,187.828,-64.257,-179.163,9.199,149.568
C05148=1121.974,187.579,-64.232,-179.166,9.196,149.568
C05149=1121.978,187.331,-64.208,-179.168,9.193,149.568
C05150=1121.982,187.081,-64.184,-179.170,9.190,149.568
C05151=1121.987,186.833,-64.160,-179.173,9.187,149.568
C05152=1121.992,186.584,-64.136,-179.175,9.184,149.568
C05153=1121.997,186.335,-64.112,-179.178,9.182,149.568
C05154=1122.001,186.087,-64.088,-179.180,9.179,149.568
C05155=1122.005,185.873,-64.067,-179.183,9.176,149.568
C05156=1122.009,185.659,-64.046,-179.185,9.174,149.568
C05157=1122.012,185.445,-64.026,-179.186,9.171,149.568
C05158=1122.016,185.231,-64.005,-179.188,9.169,149.568
C05159=1122.020,185.017,-63.984,-179.191,9.166,149.568
C05160=1122.024,184.803,-63.964,-179.193,9.164,149.568
C05161=1122.028,184.589,-63.943,-179.195,9.161,149.568
C05162=1122.032,184.375,-63.923,-179.198,9.159,149.568
C05163=1122.036,184.126,-63.898,-179.200,9.155,149.568
C05164=1122.041,183.877,-63.875,-179.203,9.152,149.568
C05165=1122.045,183.629,-63.851,-179.205,9.149,149.568
C05166=1122.050,183.380,-63.827,-179.208,9.146,149.568
C05167=1122.055,183.131,-63.803,-179.210,9.143,149.568
C05168=1122.060,182.882,-63.779,-179.213,9.140,149.568
C05169=1122.064,182.634,-63.755,-179.216,9.137,149.568
C05170=1122.069,182.385,-63.732,-179.218,9.134,149.568
C05171=1122.073,182.135,-63.707,-179.221,9.131,149.568
C05172=1122.077,181.886,-63.684,-179.223,9.128,149.568
C05173=1122.082,181.638,-63.660,-179.226,9.125,149.568
C05174=1122.086,181.389,-63.637,-179.229,9.121,149.568
C05175=1122.091,181.141,-63.613,-179.232,9.118,149.568
C05176=1122.095,180.892,-63.589,-179.234,9.115,149.568
C05177=1122.100,180.643,-63.565,-179.237,9.112,149.568
C05178=1122.105,180.394,-63.542,-179.240,9.108,149.568
C05179=1122.109,180.146,-63.518,-179.243,9.105,149.568
C05180=1122.114,179.897,-63.494,-179.246,9.102,149.568
C05181=1122.118,179.648,-63.471,-179.249,9.098,149.568
C05182=1122.123,179.399,-63.447,-179.251,9.095,149.568
C05183=1122.127,179.150,-63.424,-179.254,9.092,149.568
C05184=1122.132,178.900,-63.400,-179.256,9.089,149.568
C05185=1122.136,178.652,-63.376,-179.258,9.086,149.568
C05186=1122.141,178.403,-63.352,-179.260,9.083,149.568
C05187=1122.145,178.154,-63.329,-179.262,9.081,149.568
C05188=1122.150,177.906,-63.305,-179.264,9.077,149.567
C05189=1122.154,177.656,-63.282,-179.267,9.074,149.567
C05190=1122.159,177.407,-63.258,-179.269,9.072,149.567
C05191=1122.164,177.158,-63.235,-179.271,9.068,149.567
C05192=1122.168,176.910,-63.211,-179.273,9.065,149.567
C05193=1122.173,176.661,-63.187,-179.275,9.063,149.567
C05194=1122.178,176.412,-63.164,-179.277,9.060,149.567
C05195=1122.182,176.163,-63.141,-179.279,9.057,149.567
C05196=1122.186,175.914,-63.118,-179.282,9.054,149.567
C05197=1122.191,175.666,-63.094,-179.284,9.051,149.566
C05198=1122.195,175.417,-63.071,-179.286,9.048,149.566
C05199=1122.201,175.168,-63.048,-179.288,9.045,149.566
C05200=1122.205,174.919,-63.024,-179.290,9.042,149.566
C05201=1122.210,174.670,-63.001,-179.292,9.039,149.566
C05202=1122.214,174.422,-62.978,-179.295,9.036,149.566
C05203=1122.219,174.173,-62.955,-179.297,9.033,149.566
C05204=1122.223,173.924,-62.931,-179.299,9.030,149.566
C05205=1122.228,173.675,-62.907,-179.301,9.027,149.566
C05206=1122.233,173.426,-62.884,-179.304,9.024,149.566
C05207=1122.236,173.177,-62.861,-179.306,9.021,149.565
C05208=1122.241,172.928,-62.838,-179.308,9.018,149.565
C05209=1122.246,172.679,-62.814,-179.310,9.015,149.565
C05210=1122.251,172.430,-62.791,-179.312,9.012,149.565
C05211=1122.254,172.217,-62.771,-179.314,9.009,149.565
C05212=1122.259,172.002,-62.752,-179.316,9.007,149.565
C05213=1122.262,171.788,-62.731,-179.319,9.004,149.565
C05214=1122.266,171.574,-62.712,-179.320,9.001,149.565
C05215=1122.271,171.361,-62.691,-179.322,8.999,149.565
C05216=1122.275,171.146,-62.672,-179.324,8.997,149.565
C05217=1122.278,170.932,-62.652,-179.326,8.994,149.565
C05218=1122.282,170.718,-62.632,-179.328,8.991,149.564
C05219=1122.286,170.469,-62.609,-179.330,8.989,149.564
C05220=1122.291,170.220,-62.585,-179.332,8.985,149.564
C05221=1122.297,169.971,-62.563,-179.335,8.982,149.564
C05222=1122.301,169.723,-62.540,-179.337,8.979,149.564
C05223=1122.305,169.474,-62.517,-179.339,8.976,149.564
C05224=1122.310,169.225,-62.494,-179.341,8.973,149.564
C05225=1122.314,168.976,-62.471,-179.343,8.970,149.564
C05226=1122.319,168.727,-62.448,-179.346,8.967,149.564
C05227=1122.324,168.479,-62.425,-179.349,8.964,149.564
C05228=1122.328,168.229,-62.403,-179.351,8.961,149.564
C05229=1122.333,167.980,-62.379,-179.353,8.958,149.563
C05230=1122.338,167.731,-62.356,-179.355,8.955,149.563
C05231=1122.342,167.482,-62.333,-179.358,8.952,149.563
C05232=1122.347,167.234,-62.310,-179.360,8.948,149.563
C05233=1122.351,166.985,-62.288,-179.362,8.945,149.563
C05234=1122.356,166.736,-62.265,-179.365,8.942,149.563
C05235=1122.361,166.487,-62.241,-179.367,8.938,149.563
C05236=1122.365,166.238,-62.219,-179.369,8.936,149.563
C05237=1122.370,165.989,-62.196,-179.371,8.933,149.563
C05238=1122.374,165.740,-62.173,-179.374,8.930,149.563
C05239=1122.379,165.491,-62.150,-179.376,8.926,149.562
C05240=1122.384,165.242,-62.127,-179.378,8.923,149.562
C05241=1122.388,164.994,-62.105,-179.381,8.920,149.562
C05242=1122.393,164.745,-62.082,-179.383,8.917,149.562
C05243=1122.397,164.495,-62.060,-179.385,8.914,149.562
C05244=1122.402,164.246,-62.036,-179.388,8.911,149.562
C05245=1122.407,163.998,-62.014,-179.390,8.907,149.562
C05246=1122.412,163.749,-61.991,-179.393,8.904,149.562
C05247=1122.416,163.500,-61.969,-179.395,8.901,149.562
C05248=1122.420,163.251,-61.947,-179.397,8.897,149.562
C05249=1122.425,163.002,-61.923,-179.399,8.895,149.562
C05250=1122.429,162.753,-61.901,-179.402,8.892,149.562
C05251=1122.434,162.504,-61.878,-179.404,8.888,149.561
C05252=1122.439,162.255,-61.856,-179.406,8.885,149.561
C05253=1122.444,162.006,-61.833,-179.409,8.882,149.561
C05254=1122.448,161.757,-61.811,-179.411,8.879,149.561
C05255=1122.453,161.509,-61.789,-179.413,8.876,149.561
C05256=1122.458,161.259,-61.766,-179.416,8.872,149.561
C05257=1122.462,161.010,-61.743,-179.418,8.869,149.561
C05258=1122.467,160.761,-61.721,-179.420,8.866,149.561
C05259=1122.471,160.513,-61.698,-179.423,8.862,149.560
C05260=1122.475,160.263,-61.676,-179.426,8.859,149.560
C05261=1122.481,160.015,-61.653,-179.428,8.855,149.560
C05262=1122.485,159.766,-61.631,-179.430,8.852,149.560
C05263=1122.489,159.516,-61.609,-179.433,8.849,149.560
C05264=1122.494,159.268,-61.586,-179.435,8.845,149.560
C05265=1122.499,159.019,-61.564,-179.437,8.842,149.560
C05266=1122.504,158.770,-61.542,-179.440,8.839,149.560
C05267=1122.507,158.556,-61.522,-179.441,8.836,149.560
C05268=1122.511,158.342,-61.503,-179.444,8.833,149.559
C05269=1122.515,158.127,-61.484,-179.446,8.830,149.559
C05270=1122.519,157.913,-61.465,-179.448,8.827,149.559
C05271=1122.523,157.699,-61.446,-179.450,8.824,149.559
C05272=1122.527,157.485,-61.427,-179.452,8.822,149.559
C05273=1122.531,157.271,-61.408,-179.454,8.819,149.559
C05274=1122.535,157.056,-61.388,-179.456,8.816,149.559
C05275=1122.540,156.808,-61.366,-179.458,8.813,149.559
C05276=1122.545,156.559,-61.343,-179.462,8.809,149.559
C05277=1122.549,156.309,-61.321,-179.464,8.805,149.558
C05278=1122.554,156.061,-61.300,-179.466,8.802,149.558
C05279=1122.558,155.811,-61.278,-179.468,8.799,149.558
C05280=1122.563,155.563,-61.255,-179.471,8.796,149.558
C05281=1122.568,155.314,-61.233,-179.473,8.792,149.558
C05282=1122.573,155.065,-61.211,-179.476,8.788,149.558
C05283=1122.577,154.816,-61.189,-179.478,8.785,149.558
C05284=1122.582,154.567,-61.167,-179.480,8.781,149.557
C05285=1122.586,154.318,-61.145,-179.483,8.778,149.557
C05286=1122.592,154.069,-61.123,-179.485,8.774,149.557
C05287=1122.596,153.820,-61.101,-179.488,8.771,149.557
C05288=1122.601,153.572,-61.078,-179.490,8.767,149.557
C05289=1122.605,153.322,-61.056,-179.493,8.764,149.557
C05290=1122.610,153.074,-61.035,-179.495,8.760,149.557
C05291=1122.614,152.824,-61.013,-179.497,8.756,149.556
C05292=1122.619,152.576,-60.991,-179.500,8.753,149.556
C05293=1122.623,152.326,-60.969,-179.503,8.749,149.556
C05294=1122.629,152.077,-60.947,-179.505,8.746,149.556
C05295=1122.633,151.828,-60.925,-179.507,8.743,149.556
C05296=1122.638,151.579,-60.903,-179.509,8.739,149.556
C05297=1122.642,151.330,-60.881,-179.512,8.735,149.556
C05298=1122.647,151.081,-60.860,-179.514,8.732,149.555
C05299=1122.652,150.832,-60.838,-179.517,8.727,149.555
C05300=1122.657,150.583,-60.816,-179.520,8.724,149.555
C05301=1122.661,150.334,-60.795,-179.522,8.721,149.555
C05302=1122.666,150.085,-60.772,-179.524,8.717,149.555
C05303=1122.671,149.836,-60.751,-179.527,8.713,149.554
C05304=1122.675,149.587,-60.729,-179.529,8.710,149.554
C05305=1122.680,149.338,-60.707,-179.532,8.706,149.554
C05306=1122.685,149.089,-60.686,-179.534,8.702,149.554
C05307=1122.689,148.840,-60.664,-179.537,8.698,149.554
C05308=1122.694,148.591,-60.642,-179.539,8.695,149.554
C05309=1122.699,148.342,-60.621,-179.542,8.691,149.553
C05310=1122.703,148.093,-60.599,-179.544,8.687,149.553
C05311=1122.708,147.844,-60.578,-179.546,8.684,149.553
C05312=1122.713,147.595,-60.556,-179.549,8.680,149.553
C05313=1122.717,147.346,-60.534,-179.551,8.676,149.553
C05314=1122.722,147.097,-60.513,-179.554,8.672,149.552
C05315=1122.727,146.848,-60.492,-179.556,8.668,149.552
C05316=1122.731,146.599,-60.470,-179.559,8.664,149.552
C05317=1122.736,146.350,-60.448,-179.561,8.661,149.552
C05318=1122.741,146.101,-60.427,-179.564,8.656,149.551
C05319=1122.745,145.851,-60.405,-179.566,8.652,149.551
C05320=1122.750,145.603,-60.383,-179.569,8.649,149.551
C05321=1122.755,145.354,-60.363,-179.571,8.645,149.551
C05322=1122.759,145.105,-60.341,-179.574,8.641,149.551
C05323=1122.764,144.890,-60.323,-179.575,8.638,149.550
C05324=1122.767,144.677,-60.305,-179.576,8.635,149.550
C05325=1122.772,144.462,-60.286,-179.577,8.632,149.550
C05326=1122.776,144.248,-60.267,-179.578,8.630,149.549
C05327=1122.779,144.033,-60.249,-179.580,8.627,149.549
C05328=1122.784,143.820,-60.231,-179.581,8.624,149.549
C05329=1122.788,143.605,-60.213,-179.582,8.621,149.549
C05330=1122.792,143.390,-60.194,-179.584,8.618,149.548
C05331=1122.797,143.142,-60.173,-179.585,8.615,149.548
C05332=1122.801,142.892,-60.152,-179.587,8.611,149.547
C05333=1122.806,142.643,-60.130,-179.589,8.608,149.547
C05334=1122.811,142.394,-60.109,-179.590,8.604,149.547
C05335=1122.815,142.146,-60.088,-179.592,8.601,149.547
C05336=1122.820,141.896,-60.067,-179.593,8.598,149.546
C05337=1122.824,141.647,-60.045,-179.595,8.595,149.546
C05338=1122.830,141.398,-60.024,-179.596,8.591,149.545
C05339=1122.834,141.150,-60.003,-179.598,8.588,149.545
C05340=1122.838,140.900,-59.982,-179.599,8.584,149.545
C05341=1122.843,140.651,-59.960,-179.601,8.582,149.545
C05342=1122.848,140.402,-59.940,-179.603,8.578,149.544
C05343=1122.853,140.153,-59.919,-179.604,8.575,149.544
C05344=1122.858,139.904,-59.897,-179.606,8.571,149.543
C05345=1122.861,139.654,-59.876,-179.608,8.568,149.543
C05346=1122.867,139.405,-59.855,-179.609,8.565,149.543
C05347=1122.872,139.157,-59.834,-179.611,8.561,149.543
C05348=1122.876,138.908,-59.813,-179.612,8.558,149.542
C05349=1122.881,138.659,-59.792,-179.614,8.555,149.542
C05350=1122.885,138.409,-59.770,-179.615,8.551,149.541
C05351=1122.890,138.160,-59.750,-179.617,8.548,149.541
C05352=1122.895,137.911,-59.729,-179.618,8.545,149.541
C05353=1122.900,137.662,-59.707,-179.620,8.541,149.541
C05354=1122.904,137.413,-59.687,-179.622,8.538,149.540
C05355=1122.909,137.164,-59.666,-179.623,8.535,149.540
C05356=1122.914,136.916,-59.645,-179.625,8.531,149.540
C05357=1122.918,136.666,-59.624,-179.627,8.529,149.539
C05358=1122.923,136.417,-59.603,-179.628,8.525,149.539
C05359=1122.928,136.167,-59.582,-179.630,8.522,149.539
C05360=1122.933,135.918,-59.561,-179.631,8.518,149.538
C05361=1122.937,135.670,-59.540,-179.633,8.515,149.538
C05362=1122.942,135.421,-59.519,-179.635,8.512,149.538
C05363=1122.947,135.172,-59.499,-179.636,8.508,149.537
C05364=1122.952,134.922,-59.478,-179.638,8.505,149.537
C05365=1122.956,134.673,-59.457,-179.640,8.502,149.537
C05366=1122.961,134.424,-59.435,-179.642,8.498,149.537
C05367=1122.965,134.175,-59.415,-179.643,8.495,149.536
C05368=1122.970,133.926,-59.394,-179.645,8.491,149.536
C05369=1122.975,133.677,-59.374,-179.646,8.489,149.536
C05370=1122.980,133.428,-59.353,-179.648,8.485,149.535
C05371=1122.984,133.179,-59.332,-179.650,8.481,149.535
C05372=1122.989,132.930,-59.311,-179.651,8.479,149.535
C05373=1122.994,132.681,-59.291,-179.653,8.475,149.535
C05374=1122.999,132.431,-59.270,-179.655,8.472,149.534
C05375=1123.003,132.182,-59.250,-179.656,8.469,149.534
C05376=1123.009,131.933,-59.229,-179.659,8.465,149.534
C05377=1123.013,131.684,-59.208,-179.660,8.462,149.533
C05378=1123.018,131.436,-59.187,-179.662,8.458,149.533
C05379=1123.022,131.220,-59.170,-179.663,8.456,149.533
C05380=1123.026,131.006,-59.152,-179.664,8.453,149.533
C05381=1123.030,130.792,-59.134,-179.666,8.450,149.532
C05382=1123.034,130.577,-59.116,-179.667,8.448,149.532
C05383=1123.038,130.363,-59.098,-179.669,8.444,149.532
C05384=1123.042,130.149,-59.081,-179.671,8.441,149.532
C05385=1123.046,129.935,-59.063,-179.672,8.439,149.531
C05386=1123.051,129.720,-59.045,-179.673,8.436,149.531
C05387=1123.055,129.471,-59.025,-179.675,8.432,149.531
C05388=1123.060,129.223,-59.004,-179.677,8.429,149.531
C05389=1123.065,128.973,-58.983,-179.679,8.426,149.530
C05390=1123.069,128.724,-58.963,-179.681,8.422,149.530
C05391=1123.074,128.475,-58.943,-179.682,8.419,149.530
C05392=1123.079,128.225,-58.922,-179.684,8.416,149.529
C05393=1123.084,127.977,-58.902,-179.686,8.413,149.529
C05394=1123.088,127.728,-58.882,-179.687,8.409,149.529
C05395=1123.093,127.478,-58.861,-179.689,8.406,149.529
C05396=1123.098,127.229,-58.840,-179.691,8.403,149.528
C05397=1123.102,126.980,-58.820,-179.693,8.400,149.528
C05398=1123.108,126.731,-58.800,-179.694,8.396,149.528
C05399=1123.112,126.482,-58.779,-179.696,8.392,149.527
C05400=1123.116,126.233,-58.759,-179.698,8.389,149.527
C05401=1123.121,125.984,-58.739,-179.700,8.386,149.527
C05402=1123.126,125.734,-58.718,-179.702,8.382,149.527
C05403=1123.131,125.485,-58.698,-179.703,8.379,149.526
C05404=1123.135,125.236,-58.678,-179.705,8.376,149.526
C05405=1123.140,124.987,-58.657,-179.707,8.372,149.526
C05406=1123.145,124.738,-58.636,-179.708,8.369,149.525
C05407=1123.150,124.488,-58.617,-179.710,8.366,149.525
C05408=1123.154,124.239,-58.596,-179.712,8.362,149.525
C05409=1123.159,123.991,-58.576,-179.714,8.360,149.525
C05410=1123.164,123.741,-58.557,-179.716,8.356,149.525
C05411=1123.169,123.492,-58.536,-179.717,8.352,149.524
C05412=1123.173,123.243,-58.515,-179.719,8.349,149.524
C05413=1123.178,122.994,-58.496,-179.721,8.346,149.524
C05414=1123.183,122.745,-58.475,-179.723,8.342,149.523
C05415=1123.187,122.496,-58.455,-179.725,8.339,149.523
C05416=1123.193,122.246,-58.435,-179.727,8.335,149.523
C05417=1123.197,121.997,-58.414,-179.728,8.332,149.523
C05418=1123.202,121.749,-58.394,-179.730,8.329,149.522
C05419=1123.207,121.499,-58.375,-179.732,8.325,149.522
C05420=1123.211,121.250,-58.354,-179.734,8.322,149.522
C05421=1123.216,121.001,-58.335,-179.735,8.319,149.521
C05422=1123.220,120.752,-58.314,-179.737,8.315,149.521
C05423=1123.225,120.502,-58.295,-179.739,8.312,149.521
C05424=1123.231,120.253,-58.274,-179.741,8.308,149.521
C05425=1123.236,120.004,-58.254,-179.742,8.305,149.520
C05426=1123.240,119.755,-58.234,-179.745,8.302,149.520
C05427=1123.245,119.505,-58.214,-179.747,8.298,149.520
C05428=1123.249,119.256,-58.194,-179.749,8.295,149.520
C05429=1123.254,119.007,-58.174,-179.750,8.292,149.519
C05430=1123.259,118.759,-58.154,-179.752,8.288,149.519
C05431=1123.264,118.509,-58.135,-179.754,8.285,149.519
C05432=1123.268,118.260,-58.114,-179.756,8.281,149.519
C05433=1123.273,118.011,-58.095,-179.758,8.278,149.518
C05434=1123.278,117.762,-58.074,-179.759,8.275,149.518
C05435=1123.282,117.547,-58.057,-179.761,8.271,149.518
C05436=1123.286,117.333,-58.041,-179.762,8.268,149.518
C05437=1123.290,117.118,-58.023,-179.764,8.266,149.517
C05438=1123.295,116.904,-58.006,-179.766,8.262,149.517
C05439=1123.298,116.689,-57.988,-179.767,8.259,149.517
C05440=1123.303,116.475,-57.972,-179.769,8.257,149.517
C05441=1123.306,116.260,-57.955,-179.771,8.253,149.516
C05442=1123.310,116.046,-57.938,-179.772,8.250,149.516
C05443=1123.315,115.797,-57.918,-179.774,8.247,149.516
C05444=1123.320,115.548,-57.899,-179.776,8.244,149.516
C05445=1123.325,115.299,-57.879,-179.777,8.240,149.515
C05446=1123.330,115.049,-57.859,-179.779,8.237,149.515
C05447=1123.334,114.800,-57.839,-179.782,8.233,149.515
C05448=1123.340,114.551,-57.820,-179.784,8.230,149.515
C05449=1123.344,114.302,-57.800,-179.785,8.226,149.514
C05450=1123.349,114.052,-57.780,-179.787,8.222,149.514
C05451=1123.354,113.804,-57.761,-179.789,8.219,149.514
C05452=1123.359,113.554,-57.741,-179.791,8.216,149.514
C05453=1123.363,113.305,-57.721,-179.793,8.213,149.513
C05454=1123.368,113.056,-57.702,-179.794,8.209,149.513
C05455=1123.373,112.807,-57.682,-179.797,8.205,149.513
C05456=1123.378,112.557,-57.663,-179.799,8.202,149.512
C05457=1123.383,112.308,-57.643,-179.801,8.198,149.512
C05458=1123.388,112.059,-57.624,-179.802,8.194,149.512
